LIN {X 0,Y 314.91,Z 685.03,A -85,B 0,C 180,E1 14211.742,E2 14211.742} C_VEL
LIN {X 0,Y 315.552,Z 685.03,A -85,B 0,C 180,E1 14220.006,E2 14220.006} C_VEL
LIN {X 0,Y 314.856,Z 685.03,A -85,B 0,C 180,E1 14228.272,E2 14228.272} C_VEL
LIN {X 0,Y 314.303,Z 685.03,A -85,B 0,C 180,E1 14236.747,E2 14236.747} C_VEL
LIN {X 0,Y 313.867,Z 685.03,A -85,B 0,C 180,E1 14244.013,E2 14244.013} C_VEL
LIN {X 0,Y 313.657,Z 685.474,A -85,B 0,C 180,E1 14251.561,E2 14251.561} C_VEL
LIN {X 0,Y 320.452,Z 702.79,A -85,B 0,C 180,E1 14254.351,E2 14254.351} C_VEL
LIN {X 0,Y 344.549,Z 753.186,A -85,B 0,C 180,E1 14259.732,E2 14259.732} C_VEL
LIN {X 0,Y 358.041,Z 788.652,A -85,B 0,C 180,E1 14263.338,E2 14263.338} C_VEL
LIN {X 0,Y 350.721,Z 828.357,A -85,B 0,C 180,E1 14265.87,E2 14265.87} C_VEL
LIN {X 0,Y 342.562,Z 865.255,A -85,B 0,C 180,E1 14269.272,E2 14269.272} C_VEL
LIN {X 0,Y 334.419,Z 899.619,A -85,B 0,C 180,E1 14273.687,E2 14273.687} C_VEL
LIN {X 0,Y 326.94,Z 930.331,A -85,B 0,C 180,E1 14279.119,E2 14279.119} C_VEL
LIN {X 0,Y 321.25,Z 955.655,A -85,B 0,C 180,E1 14285.339,E2 14285.339} C_VEL
LIN {X 0,Y 317.975,Z 973.935,A -85,B 0,C 180,E1 14291.651,E2 14291.651} C_VEL
LIN {X 0,Y 316.694,Z 986.498,A -85,B 0,C 180,E1 14298.102,E2 14298.102} C_VEL
LIN {X 0,Y 316.54,Z 993.494,A -85,B 0,C 180,E1 14304.533,E2 14304.533} C_VEL
LIN {X 0,Y 316.69,Z 995.183,A -85,B 0,C 180,E1 14310.004,E2 14310.004} C_VEL
LIN {X 0,Y 316.59,Z 992.89,A -85,B 0,C 180,E1 14315.475,E2 14315.475} C_VEL
LIN {X 0,Y 316.815,Z 985.329,A -85,B 0,C 180,E1 14321.838,E2 14321.838} C_VEL
LIN {X 0,Y 318.156,Z 971.681,A -85,B 0,C 180,E1 14328.447,E2 14328.447} C_VEL
LIN {X 0,Y 321.438,Z 951.786,A -85,B 0,C 180,E1 14334.999,E2 14334.999} C_VEL
LIN {X 0,Y 327.008,Z 926.051,A -85,B 0,C 180,E1 14341.158,E2 14341.158} C_VEL
LIN {X 0,Y 335.591,Z 892.049,A -85,B 0,C 180,E1 14347.18,E2 14347.18} C_VEL
LIN {X 0,Y 337.508,Z 885.124,A -85,B 0,C 180,E1 14348.196,E2 14348.196} C_VEL
LIN {X 0,Y 337.867,Z 872.8,A -85,B 0,C 180,E1 14350.32,E2 14350.32} C_VEL
LIN {X 0,Y 338.147,Z 861.845,A -85,B 0,C 180,E1 14352.148,E2 14352.148} C_VEL
LIN {X 0,Y 338.618,Z 860.138,A -85,B 0,C 180,E1 14352.366,E2 14352.366} C_VEL
LIN {X 0,Y 352.636,Z 816.47,A -85,B 0,C 180,E1 14356.882,E2 14356.882} C_VEL
LIN {X 0,Y 360.703,Z 791.738,A -85,B 0,C 180,E1 14358.863,E2 14358.863} C_VEL
LIN {X 0,Y 364.085,Z 771.223,A -85,B 0,C 180,E1 14361.96,E2 14361.96} C_VEL
LIN {X 0,Y 362.599,Z 769.841,A -85,B 0,C 180,E1 14364.361,E2 14364.361} C_VEL
LIN {X 0,Y 362.059,Z 771.868,A -85,B 0,C 180,E1 14366.312,E2 14366.312} C_VEL
LIN {X 0,Y 346.456,Z 811.757,A -85,B 0,C 180,E1 14369.757,E2 14369.757} C_VEL
LIN {X 0,Y 336.821,Z 840.977,A -85,B 0,C 180,E1 14373.38,E2 14373.38} C_VEL
LIN {X 0,Y 328.963,Z 862.947,A -85,B 0,C 180,E1 14377.403,E2 14377.403} C_VEL
LIN {X 0,Y 321.914,Z 880.59,A -85,B 0,C 180,E1 14382.256,E2 14382.256} C_VEL
LIN {X 0,Y 316.885,Z 891.625,A -85,B 0,C 180,E1 14387.145,E2 14387.145} C_VEL
LIN {X 0,Y 313.836,Z 897.239,A -85,B 0,C 180,E1 14391.701,E2 14391.701} C_VEL
LIN {X 0,Y 311.784,Z 898.859,A -85,B 0,C 180,E1 14397.22,E2 14397.22} C_VEL
LIN {X 0,Y 311.166,Z 894.893,A -85,B 0,C 180,E1 14402.773,E2 14402.773} C_VEL
LIN {X 0,Y 311.633,Z 885.117,A -85,B 0,C 180,E1 14408.346,E2 14408.346} C_VEL
LIN {X 0,Y 313.435,Z 869.481,A -85,B 0,C 180,E1 14413.567,E2 14413.567} C_VEL
LIN {X 0,Y 316.293,Z 848.979,A -85,B 0,C 180,E1 14418.112,E2 14418.112} C_VEL
LIN {X 0,Y 319.772,Z 823.229,A -85,B 0,C 180,E1 14421.989,E2 14421.989} C_VEL
LIN {X 0,Y 322.925,Z 794.302,A -85,B 0,C 180,E1 14424.861,E2 14424.861} C_VEL
LIN {X 0,Y 325.253,Z 762.343,A -85,B 0,C 180,E1 14426.77,E2 14426.77} C_VEL
LIN {X 0,Y 325.571,Z 741.227,A -85,B 0,C 180,E1 14427.634,E2 14427.634} C_VEL
LIN {X 0,Y 308.112,Z 692.452,A -85,B 0,C 180,E1 14431.358,E2 14431.358} C_VEL
LIN {X 0,Y 305.675,Z 685.03,A -85,B 0,C 180,E1 14432.04,E2 14432.04} C_VEL
LIN {X 0,Y 305.44,Z 685.03,A -85,B 0,C 180,E1 14439.948,E2 14439.948} C_VEL
LIN {X 0,Y 305.597,Z 685.776,A -85,B 0,C 180,E1 14445.292,E2 14445.292} C_VEL
LIN {X 0,Y 308.509,Z 691.107,A -85,B 0,C 180,E1 14446.016,E2 14446.016} C_VEL
LIN {X 0,Y 327.842,Z 726.86,A -85,B 0,C 180,E1 14450.419,E2 14450.419} C_VEL
LIN {X 0,Y 337.738,Z 754.456,A -85,B 0,C 180,E1 14453.52,E2 14453.52} C_VEL
LIN {X 0,Y 340.064,Z 767.182,A -85,B 0,C 180,E1 14454.899,E2 14454.899} C_VEL
LIN {X 0,Y 334.973,Z 797.319,A -85,B 0,C 180,E1 14457.653,E2 14457.653} C_VEL
LIN {X 0,Y 329.004,Z 824.07,A -85,B 0,C 180,E1 14461.239,E2 14461.239} C_VEL
LIN {X 0,Y 323.053,Z 846.325,A -85,B 0,C 180,E1 14465.482,E2 14465.482} C_VEL
LIN {X 0,Y 317.303,Z 865.927,A -85,B 0,C 180,E1 14470.911,E2 14470.911} C_VEL
LIN {X 0,Y 313.335,Z 879.686,A -85,B 0,C 180,E1 14476.771,E2 14476.771} C_VEL
LIN {X 0,Y 311.078,Z 888.192,A -85,B 0,C 180,E1 14483.03,E2 14483.03} C_VEL
LIN {X 0,Y 310.44,Z 891.269,A -85,B 0,C 180,E1 14489.996,E2 14489.996} C_VEL
LIN {X 0,Y 310.948,Z 888.611,A -85,B 0,C 180,E1 14496.334,E2 14496.334} C_VEL
LIN {X 0,Y 313.064,Z 880.748,A -85,B 0,C 180,E1 14502.524,E2 14502.524} C_VEL
LIN {X 0,Y 316.507,Z 868.508,A -85,B 0,C 180,E1 14508.075,E2 14508.075} C_VEL
LIN {X 0,Y 321.859,Z 850.589,A -85,B 0,C 180,E1 14513.391,E2 14513.391} C_VEL
LIN {X 0,Y 328.127,Z 827.373,A -85,B 0,C 180,E1 14518.114,E2 14518.114} C_VEL
LIN {X 0,Y 334.275,Z 800.831,A -85,B 0,C 180,E1 14521.841,E2 14521.841} C_VEL
LIN {X 0,Y 339.405,Z 771.117,A -85,B 0,C 180,E1 14524.694,E2 14524.694} C_VEL
LIN {X 0,Y 339.697,Z 763.15,A -85,B 0,C 180,E1 14525.388,E2 14525.388} C_VEL
LIN {X 0,Y 331.408,Z 735.367,A -85,B 0,C 180,E1 14528.517,E2 14528.517} C_VEL
LIN {X 0,Y 316.791,Z 705.665,A -85,B 0,C 180,E1 14531.941,E2 14531.941} C_VEL
LIN {X 0,Y 305.58,Z 685.941,A -85,B 0,C 180,E1 14534.578,E2 14534.578} C_VEL
LIN {X 0,Y 305.491,Z 685.03,A -85,B 0,C 180,E1 14534.816,E2 14534.816} C_VEL
LIN {X 0,Y 305.405,Z 685.03,A -85,B 0,C 180,E1 14542.234,E2 14542.234} C_VEL
LIN {X 0,Y 305.731,Z 685.03,A -85,B 0,C 180,E1 14550.434,E2 14550.434} C_VEL
LIN {X 0,Y 306.036,Z 685.03,A -85,B 0,C 180,E1 14556.776,E2 14556.776} C_VEL
LIN {X 0,Y 306.448,Z 685.03,A -85,B 0,C 180,E1 14562.824,E2 14562.824} C_VEL
LIN {X 0,Y 306.846,Z 685.03,A -85,B 0,C 180,E1 14569.588,E2 14569.588} C_VEL
LIN {X 0,Y 307.396,Z 685.03,A -85,B 0,C 180,E1 14577.193,E2 14577.193} C_VEL
LIN {X 0,Y 307.447,Z 685.03,A -85,B 0,C 180,E1 14582.819,E2 14582.819} C_VEL
LIN {X 0,Y 306.722,Z 685.03,A -85,B 0,C 180,E1 14591.355,E2 14591.355} C_VEL
LIN {X 0,Y 306.323,Z 685.03,A -85,B 0,C 180,E1 14597.197,E2 14597.197} C_VEL
LIN {X 0,Y 306.014,Z 685.03,A -85,B 0,C 180,E1 14603.239,E2 14603.239} C_VEL
LIN {X 0,Y 305.747,Z 685.427,A -85,B 0,C 180,E1 14610.369,E2 14610.369} C_VEL
LIN {X 0,Y 312.127,Z 701.796,A -85,B 0,C 180,E1 14613.058,E2 14613.058} C_VEL
LIN {X 0,Y 335.006,Z 749.372,A -85,B 0,C 180,E1 14618.375,E2 14618.375} C_VEL
LIN {X 0,Y 349.645,Z 785.813,A -85,B 0,C 180,E1 14622.259,E2 14622.259} C_VEL
LIN {X 0,Y 350.911,Z 791.551,A -85,B 0,C 180,E1 14622.803,E2 14622.803} C_VEL
LIN {X 0,Y 343.248,Z 831.026,A -85,B 0,C 180,E1 14625.448,E2 14625.448} C_VEL
LIN {X 0,Y 334.145,Z 870.49,A -85,B 0,C 180,E1 14629.31,E2 14629.31} C_VEL
LIN {X 0,Y 325.544,Z 905.238,A -85,B 0,C 180,E1 14634.136,E2 14634.136} C_VEL
LIN {X 0,Y 318.201,Z 934.458,A -85,B 0,C 180,E1 14639.747,E2 14639.747} C_VEL
LIN {X 0,Y 313.124,Z 956.64,A -85,B 0,C 180,E1 14645.558,E2 14645.558} C_VEL
LIN {X 0,Y 309.963,Z 974.481,A -85,B 0,C 180,E1 14652.092,E2 14652.092} C_VEL
LIN {X 0,Y 308.835,Z 986.462,A -85,B 0,C 180,E1 14658.733,E2 14658.733} C_VEL
LIN {X 0,Y 308.712,Z 992.233,A -85,B 0,C 180,E1 14664.394,E2 14664.394} C_VEL
LIN {X 0,Y 308.877,Z 993.977,A -85,B 0,C 180,E1 14670.004,E2 14670.004} C_VEL
LIN {X 0,Y 308.762,Z 991.696,A -85,B 0,C 180,E1 14675.614,E2 14675.614} C_VEL
LIN {X 0,Y 308.927,Z 985.403,A -85,B 0,C 180,E1 14681.272,E2 14681.272} C_VEL
LIN {X 0,Y 310.144,Z 972.746,A -85,B 0,C 180,E1 14687.957,E2 14687.957} C_VEL
LIN {X 0,Y 313.523,Z 952.562,A -85,B 0,C 180,E1 14695.05,E2 14695.05} C_VEL
LIN {X 0,Y 319.623,Z 926.044,A -85,B 0,C 180,E1 14701.694,E2 14701.694} C_VEL
LIN {X 0,Y 328.624,Z 892.919,A -85,B 0,C 180,E1 14707.805,E2 14707.805} C_VEL
LIN {X 0,Y 338.618,Z 860.138,A -85,B 0,C 180,E1 14712.366,E2 14712.366} C_VEL
LIN {X 0,Y 340.112,Z 847.359,A -85,B 0,C 180,E1 14714.385,E2 14714.385} C_VEL
LIN {X 0,Y 341.457,Z 836.061,A -85,B 0,C 180,E1 14716.115,E2 14716.115} C_VEL
LIN {X 0,Y 342.022,Z 834.288,A -85,B 0,C 180,E1 14716.308,E2 14716.308} C_VEL
LIN {X 0,Y 356.359,Z 794.468,A -85,B 0,C 180,E1 14719.879,E2 14719.879} C_VEL
LIN {X 0,Y 360.175,Z 777.996,A -85,B 0,C 180,E1 14722.415,E2 14722.415} C_VEL
LIN {X 0,Y 358.705,Z 777.781,A -85,B 0,C 180,E1 14725.392,E2 14725.392} C_VEL
LIN {X 0,Y 341.73,Z 816.303,A -85,B 0,C 180,E1 14728.926,E2 14728.926} C_VEL
LIN {X 0,Y 330.611,Z 845.629,A -85,B 0,C 180,E1 14732.839,E2 14732.839} C_VEL
LIN {X 0,Y 321.592,Z 868.061,A -85,B 0,C 180,E1 14737.32,E2 14737.32} C_VEL
LIN {X 0,Y 314.828,Z 883.244,A -85,B 0,C 180,E1 14741.842,E2 14741.842} C_VEL
LIN {X 0,Y 308.974,Z 894.716,A -85,B 0,C 180,E1 14747.442,E2 14747.442} C_VEL
LIN {X 0,Y 306.241,Z 899.036,A -85,B 0,C 180,E1 14751.493,E2 14751.493} C_VEL
LIN {X 0,Y 304.036,Z 900.353,A -85,B 0,C 180,E1 14757.149,E2 14757.149} C_VEL
LIN {X 0,Y 303.375,Z 896.076,A -85,B 0,C 180,E1 14762.844,E2 14762.844} C_VEL
LIN {X 0,Y 303.865,Z 885.986,A -85,B 0,C 180,E1 14768.561,E2 14768.561} C_VEL
LIN {X 0,Y 305.793,Z 870.096,A -85,B 0,C 180,E1 14773.912,E2 14773.912} C_VEL
LIN {X 0,Y 308.745,Z 849.486,A -85,B 0,C 180,E1 14778.515,E2 14778.515} C_VEL
LIN {X 0,Y 312.222,Z 824.404,A -85,B 0,C 180,E1 14782.363,E2 14782.363} C_VEL
LIN {X 0,Y 315.563,Z 795.059,A -85,B 0,C 180,E1 14785.351,E2 14785.351} C_VEL
LIN {X 0,Y 317.967,Z 763.242,A -85,B 0,C 180,E1 14787.294,E2 14787.294} C_VEL
LIN {X 0,Y 318.42,Z 743.378,A -85,B 0,C 180,E1 14788.13,E2 14788.13} C_VEL
LIN {X 0,Y 301.443,Z 695.733,A -85,B 0,C 180,E1 14791.889,E2 14791.889} C_VEL
LIN {X 0,Y 297.704,Z 685.03,A -85,B 0,C 180,E1 14792.842,E2 14792.842} C_VEL
LIN {X 0,Y 297.489,Z 685.03,A -85,B 0,C 180,E1 14801.243,E2 14801.243} C_VEL
LIN {X 0,Y 297.615,Z 685.594,A -85,B 0,C 180,E1 14803.689,E2 14803.689} C_VEL
LIN {X 0,Y 300.308,Z 690.958,A -85,B 0,C 180,E1 14804.426,E2 14804.426} C_VEL
LIN {X 0,Y 318.532,Z 722.999,A -85,B 0,C 180,E1 14808.791,E2 14808.791} C_VEL
LIN {X 0,Y 329.284,Z 749.961,A -85,B 0,C 180,E1 14811.961,E2 14811.961} C_VEL
LIN {X 0,Y 333.667,Z 768.812,A -85,B 0,C 180,E1 14814.162,E2 14814.162} C_VEL
LIN {X 0,Y 328.098,Z 800.011,A -85,B 0,C 180,E1 14817.086,E2 14817.086} C_VEL
LIN {X 0,Y 321.852,Z 826.592,A -85,B 0,C 180,E1 14820.786,E2 14820.786} C_VEL
LIN {X 0,Y 315.427,Z 849.445,A -85,B 0,C 180,E1 14825.336,E2 14825.336} C_VEL
LIN {X 0,Y 309.592,Z 868.194,A -85,B 0,C 180,E1 14830.786,E2 14830.786} C_VEL
LIN {X 0,Y 305.724,Z 880.935,A -85,B 0,C 180,E1 14836.436,E2 14836.436} C_VEL
LIN {X 0,Y 303.349,Z 889.437,A -85,B 0,C 180,E1 14842.851,E2 14842.851} C_VEL
LIN {X 0,Y 302.655,Z 892.514,A -85,B 0,C 180,E1 14849.996,E2 14849.996} C_VEL
LIN {X 0,Y 303.348,Z 889.351,A -85,B 0,C 180,E1 14857.14,E2 14857.14} C_VEL
LIN {X 0,Y 305.741,Z 880.768,A -85,B 0,C 180,E1 14863.555,E2 14863.555} C_VEL
LIN {X 0,Y 309.978,Z 866.893,A -85,B 0,C 180,E1 14869.55,E2 14869.55} C_VEL
LIN {X 0,Y 315.622,Z 848.688,A -85,B 0,C 180,E1 14874.741,E2 14874.741} C_VEL
LIN {X 0,Y 322.403,Z 824.257,A -85,B 0,C 180,E1 14879.497,E2 14879.497} C_VEL
LIN {X 0,Y 328.797,Z 796.311,A -85,B 0,C 180,E1 14883.218,E2 14883.218} C_VEL
LIN {X 0,Y 333.385,Z 766.458,A -85,B 0,C 180,E1 14885.976,E2 14885.976} C_VEL
LIN {X 0,Y 325.504,Z 738.984,A -85,B 0,C 180,E1 14889.205,E2 14889.205} C_VEL
LIN {X 0,Y 312.062,Z 710.888,A -85,B 0,C 180,E1 14892.592,E2 14892.592} C_VEL
LIN {X 0,Y 297.61,Z 685.828,A -85,B 0,C 180,E1 14896.172,E2 14896.172} C_VEL
LIN {X 0,Y 297.495,Z 685.03,A -85,B 0,C 180,E1 14904.247,E2 14904.247} C_VEL
LIN {X 0,Y 297.869,Z 685.03,A -85,B 0,C 180,E1 14912.884,E2 14912.884} C_VEL
LIN {X 0,Y 298.237,Z 685.03,A -85,B 0,C 180,E1 14919.265,E2 14919.265} C_VEL
LIN {X 0,Y 298.695,Z 685.03,A -85,B 0,C 180,E1 14925.377,E2 14925.377} C_VEL
LIN {X 0,Y 299.258,Z 685.03,A -85,B 0,C 180,E1 14934.219,E2 14934.219} C_VEL
LIN {X 0,Y 299.741,Z 685.03,A -85,B 0,C 180,E1 14940.006,E2 14940.006} C_VEL
LIN {X 0,Y 299.197,Z 685.03,A -85,B 0,C 180,E1 14945.795,E2 14945.795} C_VEL
LIN {X 0,Y 298.564,Z 685.03,A -85,B 0,C 180,E1 14954.643,E2 14954.643} C_VEL
LIN {X 0,Y 298.181,Z 685.03,A -85,B 0,C 180,E1 14960.752,E2 14960.752} C_VEL
LIN {X 0,Y 297.79,Z 685.414,A -85,B 0,C 180,E1 14969.13,E2 14969.13} C_VEL
LIN {X 0,Y 303.851,Z 700.84,A -85,B 0,C 180,E1 14971.748,E2 14971.748} C_VEL
LIN {X 0,Y 327.157,Z 749.096,A -85,B 0,C 180,E1 14977.364,E2 14977.364} C_VEL
LIN {X 0,Y 342.417,Z 787.359,A -85,B 0,C 180,E1 14981.593,E2 14981.593} C_VEL
LIN {X 0,Y 343.752,Z 794.393,A -85,B 0,C 180,E1 14982.257,E2 14982.257} C_VEL
LIN {X 0,Y 335.528,Z 834.821,A -85,B 0,C 180,E1 14985.131,E2 14985.131} C_VEL
LIN {X 0,Y 326.37,Z 872.454,A -85,B 0,C 180,E1 14989.009,E2 14989.009} C_VEL
LIN {X 0,Y 317.9,Z 905.743,A -85,B 0,C 180,E1 14993.803,E2 14993.803} C_VEL
LIN {X 0,Y 310.234,Z 935.287,A -85,B 0,C 180,E1 14999.695,E2 14999.695} C_VEL
LIN {X 0,Y 304.859,Z 958.008,A -85,B 0,C 180,E1 15005.973,E2 15005.973} C_VEL
LIN {X 0,Y 301.965,Z 974.875,A -85,B 0,C 180,E1 15012.556,E2 15012.556} C_VEL
LIN {X 0,Y 300.993,Z 985.055,A -85,B 0,C 180,E1 15018.436,E2 15018.436} C_VEL
LIN {X 0,Y 300.894,Z 990.951,A -85,B 0,C 180,E1 15024.248,E2 15024.248} C_VEL
LIN {X 0,Y 301.065,Z 992.763,A -85,B 0,C 180,E1 15030.004,E2 15030.004} C_VEL
LIN {X 0,Y 300.939,Z 990.492,A -85,B 0,C 180,E1 15035.76,E2 15035.76} C_VEL
LIN {X 0,Y 301.079,Z 984.177,A -85,B 0,C 180,E1 15041.57,E2 15041.57} C_VEL
LIN {X 0,Y 302.38,Z 971.295,A -85,B 0,C 180,E1 15048.521,E2 15048.521} C_VEL
LIN {X 0,Y 305.942,Z 951.774,A -85,B 0,C 180,E1 15055.574,E2 15055.574} C_VEL
LIN {X 0,Y 312.455,Z 925.457,A -85,B 0,C 180,E1 15062.401,E2 15062.401} C_VEL
LIN {X 0,Y 322.589,Z 891.375,A -85,B 0,C 180,E1 15068.88,E2 15068.88} C_VEL
LIN {X 0,Y 336.375,Z 850.113,A -85,B 0,C 180,E1 15074.583,E2 15074.583} C_VEL
LIN {X 0,Y 342.022,Z 834.288,A -85,B 0,C 180,E1 15076.308,E2 15076.308} C_VEL
LIN {X 0,Y 344.91,Z 821.142,A -85,B 0,C 180,E1 15078.186,E2 15078.186} C_VEL
LIN {X 0,Y 348.257,Z 807.865,A -85,B 0,C 180,E1 15079.98,E2 15079.98} C_VEL
LIN {X 0,Y 352.562,Z 796.568,A -85,B 0,C 180,E1 15081.045,E2 15081.045} C_VEL
LIN {X 0,Y 356.225,Z 784.754,A -85,B 0,C 180,E1 15082.866,E2 15082.866} C_VEL
LIN {X 0,Y 355.329,Z 784.395,A -85,B 0,C 180,E1 15084.529,E2 15084.529} C_VEL
LIN {X 0,Y 337.166,Z 821.047,A -85,B 0,C 180,E1 15088.08,E2 15088.08} C_VEL
LIN {X 0,Y 325.143,Z 848.745,A -85,B 0,C 180,E1 15092.005,E2 15092.005} C_VEL
LIN {X 0,Y 315.667,Z 869.856,A -85,B 0,C 180,E1 15096.395,E2 15096.395} C_VEL
LIN {X 0,Y 307.77,Z 885.885,A -85,B 0,C 180,E1 15101.411,E2 15101.411} C_VEL
LIN {X 0,Y 301.692,Z 896.612,A -85,B 0,C 180,E1 15106.987,E2 15106.987} C_VEL
LIN {X 0,Y 298.639,Z 900.848,A -85,B 0,C 180,E1 15111.275,E2 15111.275} C_VEL
LIN {X 0,Y 296.282,Z 901.811,A -85,B 0,C 180,E1 15117.074,E2 15117.074} C_VEL
LIN {X 0,Y 295.585,Z 897.235,A -85,B 0,C 180,E1 15122.92,E2 15122.92} C_VEL
LIN {X 0,Y 295.948,Z 888.486,A -85,B 0,C 180,E1 15128.053,E2 15128.053} C_VEL
LIN {X 0,Y 297.771,Z 873.182,A -85,B 0,C 180,E1 15133.547,E2 15133.547} C_VEL
LIN {X 0,Y 300.658,Z 853.477,A -85,B 0,C 180,E1 15138.273,E2 15138.273} C_VEL
LIN {X 0,Y 304.329,Z 828.2,A -85,B 0,C 180,E1 15142.398,E2 15142.398} C_VEL
LIN {X 0,Y 307.827,Z 799.113,A -85,B 0,C 180,E1 15145.569,E2 15145.569} C_VEL
LIN {X 0,Y 310.479,Z 767.633,A -85,B 0,C 180,E1 15147.675,E2 15147.675} C_VEL
LIN {X 0,Y 311.047,Z 744.671,A -85,B 0,C 180,E1 15148.7,E2 15148.7} C_VEL
LIN {X 0,Y 293.605,Z 695.813,A -85,B 0,C 180,E1 15152.732,E2 15152.732} C_VEL
LIN {X 0,Y 289.657,Z 685.03,A -85,B 0,C 180,E1 15153.855,E2 15153.855} C_VEL
LIN {X 0,Y 289.583,Z 685.411,A -85,B 0,C 180,E1 15161.931,E2 15161.931} C_VEL
LIN {X 0,Y 292.1,Z 690.804,A -85,B 0,C 180,E1 15162.693,E2 15162.693} C_VEL
LIN {X 0,Y 308.6,Z 718.15,A -85,B 0,C 180,E1 15166.899,E2 15166.899} C_VEL
LIN {X 0,Y 320.84,Z 745.773,A -85,B 0,C 180,E1 15170.353,E2 15170.353} C_VEL
LIN {X 0,Y 327.286,Z 770.35,A -85,B 0,C 180,E1 15173.383,E2 15173.383} C_VEL
LIN {X 0,Y 321.591,Z 801.234,A -85,B 0,C 180,E1 15176.332,E2 15176.332} C_VEL
LIN {X 0,Y 315.11,Z 827.625,A -85,B 0,C 180,E1 15180.058,E2 15180.058} C_VEL
LIN {X 0,Y 308.351,Z 850.686,A -85,B 0,C 180,E1 15184.731,E2 15184.731} C_VEL
LIN {X 0,Y 302.218,Z 869.44,A -85,B 0,C 180,E1 15190.298,E2 15190.298} C_VEL
LIN {X 0,Y 297.784,Z 883.416,A -85,B 0,C 180,E1 15196.813,E2 15196.813} C_VEL
LIN {X 0,Y 295.601,Z 890.685,A -85,B 0,C 180,E1 15202.663,E2 15202.663} C_VEL
LIN {X 0,Y 294.864,Z 893.76,A -85,B 0,C 180,E1 15209.996,E2 15209.996} C_VEL
LIN {X 0,Y 295.601,Z 890.6,A -85,B 0,C 180,E1 15217.328,E2 15217.328} C_VEL
LIN {X 0,Y 298.144,Z 882.019,A -85,B 0,C 180,E1 15223.907,E2 15223.907} C_VEL
LIN {X 0,Y 302.632,Z 868.14,A -85,B 0,C 180,E1 15230.044,E2 15230.044} C_VEL
LIN {X 0,Y 308.551,Z 849.934,A -85,B 0,C 180,E1 15235.347,E2 15235.347} C_VEL
LIN {X 0,Y 315.542,Z 825.812,A -85,B 0,C 180,E1 15240.143,E2 15240.143} C_VEL
LIN {X 0,Y 322.323,Z 797.543,A -85,B 0,C 180,E1 15243.975,E2 15243.975} C_VEL
LIN {X 0,Y 326.938,Z 768.812,A -85,B 0,C 180,E1 15246.7,E2 15246.7} C_VEL
LIN {X 0,Y 319.406,Z 741.93,A -85,B 0,C 180,E1 15249.998,E2 15249.998} C_VEL
LIN {X 0,Y 306.159,Z 713.961,A -85,B 0,C 180,E1 15253.554,E2 15253.554} C_VEL
LIN {X 0,Y 291.571,Z 690.291,A -85,B 0,C 180,E1 15257.307,E2 15257.307} C_VEL
LIN {X 0,Y 289.534,Z 685.03,A -85,B 0,C 180,E1 15258.057,E2 15258.057} C_VEL
LIN {X 0,Y 289.659,Z 685.03,A -85,B 0,C 180,E1 15266.46,E2 15266.46} C_VEL
LIN {X 0,Y 289.863,Z 685.03,A -85,B 0,C 180,E1 15272.248,E2 15272.248} C_VEL
LIN {X 0,Y 290.34,Z 685.03,A -85,B 0,C 180,E1 15279.308,E2 15279.308} C_VEL
LIN {X 0,Y 290.918,Z 685.03,A -85,B 0,C 180,E1 15288.033,E2 15288.033} C_VEL
LIN {X 0,Y 291.57,Z 685.03,A -85,B 0,C 180,E1 15297.04,E2 15297.04} C_VEL
LIN {X 0,Y 291.623,Z 685.03,A -85,B 0,C 180,E1 15302.972,E2 15302.972} C_VEL
LIN {X 0,Y 290.813,Z 685.03,A -85,B 0,C 180,E1 15311.985,E2 15311.985} C_VEL
LIN {X 0,Y 290.286,Z 685.03,A -85,B 0,C 180,E1 15320.664,E2 15320.664} C_VEL
LIN {X 0,Y 289.886,Z 685.383,A -85,B 0,C 180,E1 15327.858,E2 15327.858} C_VEL
LIN {X 0,Y 295.63,Z 699.896,A -85,B 0,C 180,E1 15330.378,E2 15330.378} C_VEL
LIN {X 0,Y 319.22,Z 748.898,A -85,B 0,C 180,E1 15336.314,E2 15336.314} C_VEL
LIN {X 0,Y 334.247,Z 786.346,A -85,B 0,C 180,E1 15340.62,E2 15340.62} C_VEL
LIN {X 0,Y 336.831,Z 795.847,A -85,B 0,C 180,E1 15341.63,E2 15341.63} C_VEL
LIN {X 0,Y 328.33,Z 835.744,A -85,B 0,C 180,E1 15344.574,E2 15344.574} C_VEL
LIN {X 0,Y 318.983,Z 872.969,A -85,B 0,C 180,E1 15348.528,E2 15348.528} C_VEL
LIN {X 0,Y 310.308,Z 905.886,A -85,B 0,C 180,E1 15353.412,E2 15353.412} C_VEL
LIN {X 0,Y 302.588,Z 934.769,A -85,B 0,C 180,E1 15359.331,E2 15359.331} C_VEL
LIN {X 0,Y 296.902,Z 958.133,A -85,B 0,C 180,E1 15366.012,E2 15366.012} C_VEL
LIN {X 0,Y 294.026,Z 974.803,A -85,B 0,C 180,E1 15372.84,E2 15372.84} C_VEL
LIN {X 0,Y 293.098,Z 985.518,A -85,B 0,C 180,E1 15379.623,E2 15379.623} C_VEL
LIN {X 0,Y 293.067,Z 989.642,A -85,B 0,C 180,E1 15384.093,E2 15384.093} C_VEL
LIN {X 0,Y 293.277,Z 991.533,A -85,B 0,C 180,E1 15390.004,E2 15390.004} C_VEL
LIN {X 0,Y 293.107,Z 989.281,A -85,B 0,C 180,E1 15395.915,E2 15395.915} C_VEL
LIN {X 0,Y 293.243,Z 982.642,A -85,B 0,C 180,E1 15402.109,E2 15402.109} C_VEL
LIN {X 0,Y 294.6,Z 970.061,A -85,B 0,C 180,E1 15409.029,E2 15409.029} C_VEL
LIN {X 0,Y 298.476,Z 950.64,A -85,B 0,C 180,E1 15416.262,E2 15416.262} C_VEL
LIN {X 0,Y 305.6,Z 924.187,A -85,B 0,C 180,E1 15423.328,E2 15423.328} C_VEL
LIN {X 0,Y 317.038,Z 889.177,A -85,B 0,C 180,E1 15430.152,E2 15430.152} C_VEL
LIN {X 0,Y 332.242,Z 848.034,A -85,B 0,C 180,E1 15435.934,E2 15435.934} C_VEL
LIN {X 0,Y 348.257,Z 807.865,A -85,B 0,C 180,E1 15439.98,E2 15439.98} C_VEL
LIN {X 0,Y 349.723,Z 801.928,A -85,B 0,C 180,E1 15440.992,E2 15440.992} C_VEL
LIN {X 0,Y 351.205,Z 793.819,A -85,B 0,C 180,E1 15443.07,E2 15443.07} C_VEL
LIN {X 0,Y 352.109,Z 791.279,A -85,B 0,C 180,E1 15443.661,E2 15443.661} C_VEL
LIN {X 0,Y 333.305,Z 824.909,A -85,B 0,C 180,E1 15447.089,E2 15447.089} C_VEL
LIN {X 0,Y 319.803,Z 852.079,A -85,B 0,C 180,E1 15451.148,E2 15451.148} C_VEL
LIN {X 0,Y 309.08,Z 873.383,A -85,B 0,C 180,E1 15455.86,E2 15455.86} C_VEL
LIN {X 0,Y 300.743,Z 888.568,A -85,B 0,C 180,E1 15460.96,E2 15460.96} C_VEL
LIN {X 0,Y 294.296,Z 898.743,A -85,B 0,C 180,E1 15466.655,E2 15466.655} C_VEL
LIN {X 0,Y 291.054,Z 902.684,A -85,B 0,C 180,E1 15471.046,E2 15471.046} C_VEL
LIN {X 0,Y 288.535,Z 903.253,A -85,B 0,C 180,E1 15476.996,E2 15476.996} C_VEL
LIN {X 0,Y 287.794,Z 898.384,A -85,B 0,C 180,E1 15482.999,E2 15482.999} C_VEL
LIN {X 0,Y 288.333,Z 887.636,A -85,B 0,C 180,E1 15489.026,E2 15489.026} C_VEL
LIN {X 0,Y 290.286,Z 872.444,A -85,B 0,C 180,E1 15494.287,E2 15494.287} C_VEL
LIN {X 0,Y 293.428,Z 851.706,A -85,B 0,C 180,E1 15499.129,E2 15499.129} C_VEL
LIN {X 0,Y 297.186,Z 826.62,A -85,B 0,C 180,E1 15503.164,E2 15503.164} C_VEL
LIN {X 0,Y 300.739,Z 797.348,A -85,B 0,C 180,E1 15506.3,E2 15506.3} C_VEL
LIN {X 0,Y 303.382,Z 765.088,A -85,B 0,C 180,E1 15508.388,E2 15508.388} C_VEL
LIN {X 0,Y 303.815,Z 746.49,A -85,B 0,C 180,E1 15509.245,E2 15509.245} C_VEL
LIN {X 0,Y 286.357,Z 697.38,A -85,B 0,C 180,E1 15513.469,E2 15513.469} C_VEL
LIN {X 0,Y 281.715,Z 685.03,A -85,B 0,C 180,E1 15514.801,E2 15514.801} C_VEL
LIN {X 0,Y 281.711,Z 685.822,A -85,B 0,C 180,E1 15520.067,E2 15520.067} C_VEL
LIN {X 0,Y 284.697,Z 691.263,A -85,B 0,C 180,E1 15521.01,E2 15521.01} C_VEL
LIN {X 0,Y 302.327,Z 720.548,A -85,B 0,C 180,E1 15525.817,E2 15525.817} C_VEL
LIN {X 0,Y 314.306,Z 747.295,A -85,B 0,C 180,E1 15529.376,E2 15529.376} C_VEL
LIN {X 0,Y 320.914,Z 772.646,A -85,B 0,C 180,E1 15532.647,E2 15532.647} C_VEL
LIN {X 0,Y 315.136,Z 802.459,A -85,B 0,C 180,E1 15535.547,E2 15535.547} C_VEL
LIN {X 0,Y 308.032,Z 830.111,A -85,B 0,C 180,E1 15539.553,E2 15539.553} C_VEL
LIN {X 0,Y 300.702,Z 853.744,A -85,B 0,C 180,E1 15544.568,E2 15544.568} C_VEL
LIN {X 0,Y 294.883,Z 870.683,A -85,B 0,C 180,E1 15549.787,E2 15549.787} C_VEL
LIN {X 0,Y 290.549,Z 883.43,A -85,B 0,C 180,E1 15555.712,E2 15555.712} C_VEL
LIN {X 0,Y 287.878,Z 891.93,A -85,B 0,C 180,E1 15562.465,E2 15562.465} C_VEL
LIN {X 0,Y 287.149,Z 894.491,A -85,B 0,C 180,E1 15566.983,E2 15566.983} C_VEL
LIN {X 0,Y 287.172,Z 894.326,A -85,B 0,C 180,E1 15573.449,E2 15573.449} C_VEL
LIN {X 0,Y 288.835,Z 888.712,A -85,B 0,C 180,E1 15580.532,E2 15580.532} C_VEL
LIN {X 0,Y 292.627,Z 877.21,A -85,B 0,C 180,E1 15587.386,E2 15587.386} C_VEL
LIN {X 0,Y 298.418,Z 860.49,A -85,B 0,C 180,E1 15593.463,E2 15593.463} C_VEL
LIN {X 0,Y 305.508,Z 838.482,A -85,B 0,C 180,E1 15598.786,E2 15598.786} C_VEL
LIN {X 0,Y 312.752,Z 812.39,A -85,B 0,C 180,E1 15603.077,E2 15603.077} C_VEL
LIN {X 0,Y 319.082,Z 782.905,A -85,B 0,C 180,E1 15606.374,E2 15606.374} C_VEL
LIN {X 0,Y 320.633,Z 771.591,A -85,B 0,C 180,E1 15607.392,E2 15607.392} C_VEL
LIN {X 0,Y 313.14,Z 744.192,A -85,B 0,C 180,E1 15610.905,E2 15610.905} C_VEL
LIN {X 0,Y 300.403,Z 717.207,A -85,B 0,C 180,E1 15614.538,E2 15614.538} C_VEL
LIN {X 0,Y 284.194,Z 690.862,A -85,B 0,C 180,E1 15618.985,E2 15618.985} C_VEL
LIN {X 0,Y 281.738,Z 685.987,A -85,B 0,C 180,E1 15619.777,E2 15619.777} C_VEL
LIN {X 0,Y 281.639,Z 685.03,A -85,B 0,C 180,E1 15620.001,E2 15620.001} C_VEL
LIN {X 0,Y 281.762,Z 685.03,A -85,B 0,C 180,E1 15628.965,E2 15628.965} C_VEL
LIN {X 0,Y 282.213,Z 685.03,A -85,B 0,C 180,E1 15638.029,E2 15638.029} C_VEL
LIN {X 0,Y 282.739,Z 685.03,A -85,B 0,C 180,E1 15644.531,E2 15644.531} C_VEL
LIN {X 0,Y 283.227,Z 685.03,A -85,B 0,C 180,E1 15652.921,E2 15652.921} C_VEL
LIN {X 0,Y 283.929,Z 685.03,A -85,B 0,C 180,E1 15660.007,E2 15660.007} C_VEL
LIN {X 0,Y 283.33,Z 685.03,A -85,B 0,C 180,E1 15666.121,E2 15666.121} C_VEL
LIN {X 0,Y 282.845,Z 685.03,A -85,B 0,C 180,E1 15672.328,E2 15672.328} C_VEL
LIN {X 0,Y 282.408,Z 685.03,A -85,B 0,C 180,E1 15678.705,E2 15678.705} C_VEL
LIN {X 0,Y 281.951,Z 685.284,A -85,B 0,C 180,E1 15686.52,E2 15686.52} C_VEL
LIN {X 0,Y 287.386,Z 698.972,A -85,B 0,C 180,E1 15688.956,E2 15688.956} C_VEL
LIN {X 0,Y 311.231,Z 748.305,A -85,B 0,C 180,E1 15695.204,E2 15695.204} C_VEL
LIN {X 0,Y 326.789,Z 787.205,A -85,B 0,C 180,E1 15699.848,E2 15699.848} C_VEL
LIN {X 0,Y 329.716,Z 798.014,A -85,B 0,C 180,E1 15701.046,E2 15701.046} C_VEL
LIN {X 0,Y 321.174,Z 836.533,A -85,B 0,C 180,E1 15703.994,E2 15703.994} C_VEL
LIN {X 0,Y 311.719,Z 872.923,A -85,B 0,C 180,E1 15707.97,E2 15707.97} C_VEL
LIN {X 0,Y 302.766,Z 905.862,A -85,B 0,C 180,E1 15712.987,E2 15712.987} C_VEL
LIN {X 0,Y 295.03,Z 933.832,A -85,B 0,C 180,E1 15718.87,E2 15718.87} C_VEL
LIN {X 0,Y 289.13,Z 957.328,A -85,B 0,C 180,E1 15725.757,E2 15725.757} C_VEL
LIN {X 0,Y 286.271,Z 973.122,A -85,B 0,C 180,E1 15732.36,E2 15732.36} C_VEL
LIN {X 0,Y 285.282,Z 984.161,A -85,B 0,C 180,E1 15739.409,E2 15739.409} C_VEL
LIN {X 0,Y 285.274,Z 988.308,A -85,B 0,C 180,E1 15743.931,E2 15743.931} C_VEL
LIN {X 0,Y 285.475,Z 990.285,A -85,B 0,C 180,E1 15750.005,E2 15750.005} C_VEL
LIN {X 0,Y 285.268,Z 988.075,A -85,B 0,C 180,E1 15756.078,E2 15756.078} C_VEL
LIN {X 0,Y 285.442,Z 980.664,A -85,B 0,C 180,E1 15762.989,E2 15762.989} C_VEL
LIN {X 0,Y 286.967,Z 968.298,A -85,B 0,C 180,E1 15769.832,E2 15769.832} C_VEL
LIN {X 0,Y 291.048,Z 949.579,A -85,B 0,C 180,E1 15776.985,E2 15776.985} C_VEL
LIN {X 0,Y 298.715,Z 923.504,A -85,B 0,C 180,E1 15784.201,E2 15784.201} C_VEL
LIN {X 0,Y 311.295,Z 888.365,A -85,B 0,C 180,E1 15791.285,E2 15791.285} C_VEL
LIN {X 0,Y 328.461,Z 846.504,A -85,B 0,C 180,E1 15797.322,E2 15797.322} C_VEL
LIN {X 0,Y 347.557,Z 803.523,A -85,B 0,C 180,E1 15801.614,E2 15801.614} C_VEL
LIN {X 0,Y 351.205,Z 793.819,A -85,B 0,C 180,E1 15803.07,E2 15803.07} C_VEL
LIN {X 0,Y 349.901,Z 795.468,A -85,B 0,C 180,E1 15803.567,E2 15803.567} C_VEL
LIN {X 0,Y 339.331,Z 813.098,A -85,B 0,C 180,E1 15804.231,E2 15804.231} C_VEL
LIN {X 0,Y 321.505,Z 843.33,A -85,B 0,C 180,E1 15808.124,E2 15808.124} C_VEL
LIN {X 0,Y 307.469,Z 868.341,A -85,B 0,C 180,E1 15812.997,E2 15812.997} C_VEL
LIN {X 0,Y 296.971,Z 886.25,A -85,B 0,C 180,E1 15818.378,E2 15818.378} C_VEL
LIN {X 0,Y 289.11,Z 897.998,A -85,B 0,C 180,E1 15824.091,E2 15824.091} C_VEL
LIN {X 0,Y 284.333,Z 903.818,A -85,B 0,C 180,E1 15829.556,E2 15829.556} C_VEL
LIN {X 0,Y 281.97,Z 905.242,A -85,B 0,C 180,E1 15833.849,E2 15833.849} C_VEL
LIN {X 0,Y 280.373,Z 902.753,A -85,B 0,C 180,E1 15839.993,E2 15839.993} C_VEL
LIN {X 0,Y 280.073,Z 894.75,A -85,B 0,C 180,E1 15846.179,E2 15846.179} C_VEL
LIN {X 0,Y 281.423,Z 881.426,A -85,B 0,C 180,E1 15851.984,E2 15851.984} C_VEL
LIN {X 0,Y 284.32,Z 861.887,A -85,B 0,C 180,E1 15857.51,E2 15857.51} C_VEL
LIN {X 0,Y 288.107,Z 837.78,A -85,B 0,C 180,E1 15862.105,E2 15862.105} C_VEL
LIN {X 0,Y 291.852,Z 810.872,A -85,B 0,C 180,E1 15865.605,E2 15865.605} C_VEL
LIN {X 0,Y 295.133,Z 779.965,A -85,B 0,C 180,E1 15868.192,E2 15868.192} C_VEL
LIN {X 0,Y 296.69,Z 748.766,A -85,B 0,C 180,E1 15869.78,E2 15869.78} C_VEL
LIN {X 0,Y 279.981,Z 701.251,A -85,B 0,C 180,E1 15874.001,E2 15874.001} C_VEL
LIN {X 0,Y 273.682,Z 685.03,A -85,B 0,C 180,E1 15875.872,E2 15875.872} C_VEL
LIN {X 0,Y 273.567,Z 685.03,A -85,B 0,C 180,E1 15877.872,E2 15877.872} C_VEL
LIN {X 0,Y 275.838,Z 690.531,A -85,B 0,C 180,E1 15878.737,E2 15878.737} C_VEL
LIN {X 0,Y 282.135,Z 699.697,A -85,B 0,C 180,E1 15880.718,E2 15880.718} C_VEL
LIN {X 0,Y 298.098,Z 726.566,A -85,B 0,C 180,E1 15885.235,E2 15885.235} C_VEL
LIN {X 0,Y 308.936,Z 752.364,A -85,B 0,C 180,E1 15888.821,E2 15888.821} C_VEL
LIN {X 0,Y 314.426,Z 776.099,A -85,B 0,C 180,E1 15891.981,E2 15891.981} C_VEL
LIN {X 0,Y 308.113,Z 806.451,A -85,B 0,C 180,E1 15895.075,E2 15895.075} C_VEL
LIN {X 0,Y 300.566,Z 833.959,A -85,B 0,C 180,E1 15899.265,E2 15899.265} C_VEL
LIN {X 0,Y 293.058,Z 856.76,A -85,B 0,C 180,E1 15904.384,E2 15904.384} C_VEL
LIN {X 0,Y 286.877,Z 873.809,A -85,B 0,C 180,E1 15910.001,E2 15910.001} C_VEL
LIN {X 0,Y 282.562,Z 885.916,A -85,B 0,C 180,E1 15916.089,E2 15916.089} C_VEL
LIN {X 0,Y 280.151,Z 893.175,A -85,B 0,C 180,E1 15922.256,E2 15922.256} C_VEL
LIN {X 0,Y 279.285,Z 896.252,A -85,B 0,C 180,E1 15929.995,E2 15929.995} C_VEL
LIN {X 0,Y 280.154,Z 893.093,A -85,B 0,C 180,E1 15937.735,E2 15937.735} C_VEL
LIN {X 0,Y 283.008,Z 884.517,A -85,B 0,C 180,E1 15944.667,E2 15944.667} C_VEL
LIN {X 0,Y 288.004,Z 870.638,A -85,B 0,C 180,E1 15951.11,E2 15951.11} C_VEL
LIN {X 0,Y 294.672,Z 851.943,A -85,B 0,C 180,E1 15956.766,E2 15956.766} C_VEL
LIN {X 0,Y 302.468,Z 827.292,A -85,B 0,C 180,E1 15961.802,E2 15961.802} C_VEL
LIN {X 0,Y 309.527,Z 800.012,A -85,B 0,C 180,E1 15965.587,E2 15965.587} C_VEL
LIN {X 0,Y 314.356,Z 774.663,A -85,B 0,C 180,E1 15968.069,E2 15968.069} C_VEL
LIN {X 0,Y 307.217,Z 747.369,A -85,B 0,C 180,E1 15971.742,E2 15971.742} C_VEL
LIN {X 0,Y 294.594,Z 720.159,A -85,B 0,C 180,E1 15975.6,E2 15975.6} C_VEL
LIN {X 0,Y 279.366,Z 695.708,A -85,B 0,C 180,E1 15979.986,E2 15979.986} C_VEL
LIN {X 0,Y 275.787,Z 690.47,A -85,B 0,C 180,E1 15981.131,E2 15981.131} C_VEL
LIN {X 0,Y 273.55,Z 685.03,A -85,B 0,C 180,E1 15982.112,E2 15982.112} C_VEL
LIN {X 0,Y 273.866,Z 685.03,A -85,B 0,C 180,E1 15990.282,E2 15990.282} C_VEL
LIN {X 0,Y 274.308,Z 685.03,A -85,B 0,C 180,E1 15999.253,E2 15999.253} C_VEL
LIN {X 0,Y 275.012,Z 685.03,A -85,B 0,C 180,E1 16007.33,E2 16007.33} C_VEL
LIN {X 0,Y 275.448,Z 685.03,A -85,B 0,C 180,E1 16013.717,E2 16013.717} C_VEL
LIN {X 0,Y 276.022,Z 685.03,A -85,B 0,C 180,E1 16020.007,E2 16020.007} C_VEL
LIN {X 0,Y 275.39,Z 685.03,A -85,B 0,C 180,E1 16026.298,E2 16026.298} C_VEL
LIN {X 0,Y 274.89,Z 685.03,A -85,B 0,C 180,E1 16032.69,E2 16032.69} C_VEL
LIN {X 0,Y 274.279,Z 685.03,A -85,B 0,C 180,E1 16040.731,E2 16040.731} C_VEL
LIN {X 0,Y 274.134,Z 685.529,A -85,B 0,C 180,E1 16045.2,E2 16045.2} C_VEL
LIN {X 0,Y 279.107,Z 698.033,A -85,B 0,C 180,E1 16047.473,E2 16047.473} C_VEL
LIN {X 0,Y 302.675,Z 746.502,A -85,B 0,C 180,E1 16053.905,E2 16053.905} C_VEL
LIN {X 0,Y 318.662,Z 786.235,A -85,B 0,C 180,E1 16058.829,E2 16058.829} C_VEL
LIN {X 0,Y 322.778,Z 798.298,A -85,B 0,C 180,E1 16060.312,E2 16060.312} C_VEL
LIN {X 0,Y 313.954,Z 837.522,A -85,B 0,C 180,E1 16063.429,E2 16063.429} C_VEL
LIN {X 0,Y 303.976,Z 874.709,A -85,B 0,C 180,E1 16067.642,E2 16067.642} C_VEL
LIN {X 0,Y 294.543,Z 908.168,A -85,B 0,C 180,E1 16072.992,E2 16072.992} C_VEL
LIN {X 0,Y 286.401,Z 936.747,A -85,B 0,C 180,E1 16079.405,E2 16079.405} C_VEL
LIN {X 0,Y 280.904,Z 958.767,A -85,B 0,C 180,E1 16086.347,E2 16086.347} C_VEL
LIN {X 0,Y 278.185,Z 974.421,A -85,B 0,C 180,E1 16093.479,E2 16093.479} C_VEL
LIN {X 0,Y 277.411,Z 984.311,A -85,B 0,C 180,E1 16100.612,E2 16100.612} C_VEL
LIN {X 0,Y 277.501,Z 988.502,A -85,B 0,C 180,E1 16106.887,E2 16106.887} C_VEL
LIN {X 0,Y 277.687,Z 989.03,A -85,B 0,C 180,E1 16110.005,E2 16110.005} C_VEL
LIN {X 0,Y 277.436,Z 986.858,A -85,B 0,C 180,E1 16116.25,E2 16116.25} C_VEL
LIN {X 0,Y 277.597,Z 979.474,A -85,B 0,C 180,E1 16123.363,E2 16123.363} C_VEL
LIN {X 0,Y 279.377,Z 966.832,A -85,B 0,C 180,E1 16130.56,E2 16130.56} C_VEL
LIN {X 0,Y 284.371,Z 946.229,A -85,B 0,C 180,E1 16138.534,E2 16138.534} C_VEL
LIN {X 0,Y 293.69,Z 918.317,A -85,B 0,C 180,E1 16146.227,E2 16146.227} C_VEL
LIN {X 0,Y 307.973,Z 882.851,A -85,B 0,C 180,E1 16153.321,E2 16153.321} C_VEL
LIN {X 0,Y 326.736,Z 842.093,A -85,B 0,C 180,E1 16159.146,E2 16159.146} C_VEL
LIN {X 0,Y 345.376,Z 804.222,A -85,B 0,C 180,E1 16162.993,E2 16162.993} C_VEL
LIN {X 0,Y 345.969,Z 802.844,A -85,B 0,C 180,E1 16163.235,E2 16163.235} C_VEL
LIN {X 0,Y 339.331,Z 813.098,A -85,B 0,C 180,E1 16164.231,E2 16164.231} C_VEL
LIN {X 0,Y 336.407,Z 818.105,A -85,B 0,C 180,E1 16164.084,E2 16164.084} C_VEL
LIN {X 0,Y 330.276,Z 830.129,A -85,B 0,C 180,E1 16161.874,E2 16161.874} C_VEL
LIN {X 0,Y 309.198,Z 869.912,A -85,B 0,C 180,E1 16156.689,E2 16156.689} C_VEL
LIN {X 0,Y 291.777,Z 906.903,A -85,B 0,C 180,E1 16149.801,E2 16149.801} C_VEL
LIN {X 0,Y 280.098,Z 936.807,A -85,B 0,C 180,E1 16142.103,E2 16142.103} C_VEL
LIN {X 0,Y 273.094,Z 959.905,A -85,B 0,C 180,E1 16133.842,E2 16133.842} C_VEL
LIN {X 0,Y 270.155,Z 974.687,A -85,B 0,C 180,E1 16126.223,E2 16126.223} C_VEL
LIN {X 0,Y 269.582,Z 983.002,A -85,B 0,C 180,E1 16119.673,E2 16119.673} C_VEL
LIN {X 0,Y 269.658,Z 987.182,A -85,B 0,C 180,E1 16113.213,E2 16113.213} C_VEL
LIN {X 0,Y 269.911,Z 987.746,A -85,B 0,C 180,E1 16110.005,E2 16110.005} C_VEL
LIN {X 0,Y 269.666,Z 985.554,A -85,B 0,C 180,E1 16103.579,E2 16103.579} C_VEL
LIN {X 0,Y 269.848,Z 977.876,A -85,B 0,C 180,E1 16096.256,E2 16096.256} C_VEL
LIN {X 0,Y 271.781,Z 964.439,A -85,B 0,C 180,E1 16088.849,E2 16088.849} C_VEL
LIN {X 0,Y 276.439,Z 944.479,A -85,B 0,C 180,E1 16081.473,E2 16081.473} C_VEL
LIN {X 0,Y 283.889,Z 918.129,A -85,B 0,C 180,E1 16074.638,E2 16074.638} C_VEL
LIN {X 0,Y 293.337,Z 886.308,A -85,B 0,C 180,E1 16068.771,E2 16068.771} C_VEL
LIN {X 0,Y 303.492,Z 850.476,A -85,B 0,C 180,E1 16064.085,E2 16064.085} C_VEL
LIN {X 0,Y 313.182,Z 811.673,A -85,B 0,C 180,E1 16060.517,E2 16060.517} C_VEL
LIN {X 0,Y 315.243,Z 799.118,A -85,B 0,C 180,E1 16059.543,E2 16059.543} C_VEL
LIN {X 0,Y 301.273,Z 761.794,A -85,B 0,C 180,E1 16054.737,E2 16054.737} C_VEL
LIN {X 0,Y 282.702,Z 720.798,A -85,B 0,C 180,E1 16049.348,E2 16049.348} C_VEL
LIN {X 0,Y 267.758,Z 689.553,A -85,B 0,C 180,E1 16044.661,E2 16044.661} C_VEL
LIN {X 0,Y 266.29,Z 685.03,A -85,B 0,C 180,E1 16043.554,E2 16043.554} C_VEL
LIN {X 0,Y 266.763,Z 685.03,A -85,B 0,C 180,E1 16035.928,E2 16035.928} C_VEL
LIN {X 0,Y 267.451,Z 685.03,A -85,B 0,C 180,E1 16026.486,E2 16026.486} C_VEL
LIN {X 0,Y 268.114,Z 685.03,A -85,B 0,C 180,E1 16020.007,E2 16020.007} C_VEL
LIN {X 0,Y 267.414,Z 685.03,A -85,B 0,C 180,E1 16013.022,E2 16013.022} C_VEL
LIN {X 0,Y 266.862,Z 685.03,A -85,B 0,C 180,E1 16003.997,E2 16003.997} C_VEL
LIN {X 0,Y 266.062,Z 685.03,A -85,B 0,C 180,E1 15995.151,E2 15995.151} C_VEL
LIN {X 0,Y 265.728,Z 685.03,A -85,B 0,C 180,E1 15988.405,E2 15988.405} C_VEL
LIN {X 0,Y 265.623,Z 685.304,A -85,B 0,C 180,E1 15984.29,E2 15984.29} C_VEL
LIN {X 0,Y 267.851,Z 690.541,A -85,B 0,C 180,E1 15983.37,E2 15983.37} C_VEL
LIN {X 0,Y 270.526,Z 694.158,A -85,B 0,C 180,E1 15982.428,E2 15982.428} C_VEL
LIN {X 0,Y 286.043,Z 718.162,A -85,B 0,C 180,E1 15977.519,E2 15977.519} C_VEL
LIN {X 0,Y 298.961,Z 744.292,A -85,B 0,C 180,E1 15973.498,E2 15973.498} C_VEL
LIN {X 0,Y 306.8,Z 770.275,A -85,B 0,C 180,E1 15969.819,E2 15969.819} C_VEL
LIN {X 0,Y 307.774,Z 779.758,A -85,B 0,C 180,E1 15968.602,E2 15968.602} C_VEL
LIN {X 0,Y 301.148,Z 809.672,A -85,B 0,C 180,E1 15965.404,E2 15965.404} C_VEL
LIN {X 0,Y 293.432,Z 836.303,A -85,B 0,C 180,E1 15961.187,E2 15961.187} C_VEL
LIN {X 0,Y 285.598,Z 859.135,A -85,B 0,C 180,E1 15955.869,E2 15955.869} C_VEL
LIN {X 0,Y 278.942,Z 876.631,A -85,B 0,C 180,E1 15949.758,E2 15949.758} C_VEL
LIN {X 0,Y 274.232,Z 889.24,A -85,B 0,C 180,E1 15942.711,E2 15942.711} C_VEL
LIN {X 0,Y 272.01,Z 895.461,A -85,B 0,C 180,E1 15936.366,E2 15936.366} C_VEL
LIN {X 0,Y 271.509,Z 897.495,A -85,B 0,C 180,E1 15929.995,E2 15929.995} C_VEL
LIN {X 0,Y 272.416,Z 894.423,A -85,B 0,C 180,E1 15922.035,E2 15922.035} C_VEL
LIN {X 0,Y 275.42,Z 885.927,A -85,B 0,C 180,E1 15914.909,E2 15914.909} C_VEL
LIN {X 0,Y 280.641,Z 872.157,A -85,B 0,C 180,E1 15908.299,E2 15908.299} C_VEL
LIN {X 0,Y 287.674,Z 853.46,A -85,B 0,C 180,E1 15902.486,E2 15902.486} C_VEL
LIN {X 0,Y 295.722,Z 829.326,A -85,B 0,C 180,E1 15897.437,E2 15897.437} C_VEL
LIN {X 0,Y 303.119,Z 801.977,A -85,B 0,C 180,E1 15893.531,E2 15893.531} C_VEL
LIN {X 0,Y 308.072,Z 776.35,A -85,B 0,C 180,E1 15890.935,E2 15890.935} C_VEL
LIN {X 0,Y 301.242,Z 750.134,A -85,B 0,C 180,E1 15887.222,E2 15887.222} C_VEL
LIN {X 0,Y 288.935,Z 723.024,A -85,B 0,C 180,E1 15883.169,E2 15883.169} C_VEL
LIN {X 0,Y 272.858,Z 697.408,A -85,B 0,C 180,E1 15878.216,E2 15878.216} C_VEL
LIN {X 0,Y 267.66,Z 690.176,A -85,B 0,C 180,E1 15876.399,E2 15876.399} C_VEL
LIN {X 0,Y 268.193,Z 692.264,A -85,B 0,C 180,E1 15875.987,E2 15875.987} C_VEL
LIN {X 0,Y 284.883,Z 736.044,A -85,B 0,C 180,E1 15871.579,E2 15871.579} C_VEL
LIN {X 0,Y 289.791,Z 753.638,A -85,B 0,C 180,E1 15870.176,E2 15870.176} C_VEL
LIN {X 0,Y 286.974,Z 789.75,A -85,B 0,C 180,E1 15868.128,E2 15868.128} C_VEL
LIN {X 0,Y 283.358,Z 819.626,A -85,B 0,C 180,E1 15865.206,E2 15865.206} C_VEL
LIN {X 0,Y 279.292,Z 846.671,A -85,B 0,C 180,E1 15861.172,E2 15861.172} C_VEL
LIN {X 0,Y 275.553,Z 869.42,A -85,B 0,C 180,E1 15856.163,E2 15856.163} C_VEL
LIN {X 0,Y 272.996,Z 887.253,A -85,B 0,C 180,E1 15850.341,E2 15850.341} C_VEL
LIN {X 0,Y 272.162,Z 898.289,A -85,B 0,C 180,E1 15844.762,E2 15844.762} C_VEL
LIN {X 0,Y 272.735,Z 905.249,A -85,B 0,C 180,E1 15838.408,E2 15838.408} C_VEL
LIN {X 0,Y 274.305,Z 906.846,A -85,B 0,C 180,E1 15833.677,E2 15833.677} C_VEL
LIN {X 0,Y 278.191,Z 904.497,A -85,B 0,C 180,E1 15827.463,E2 15827.463} C_VEL
LIN {X 0,Y 284.686,Z 896.871,A -85,B 0,C 180,E1 15821.45,E2 15821.45} C_VEL
LIN {X 0,Y 294.683,Z 882.688,A -85,B 0,C 180,E1 15815.409,E2 15815.409} C_VEL
LIN {X 0,Y 307.304,Z 862.983,A -85,B 0,C 180,E1 15810.13,E2 15810.13} C_VEL
LIN {X 0,Y 323.774,Z 837.201,A -85,B 0,C 180,E1 15805.579,E2 15805.579} C_VEL
LIN {X 0,Y 336.53,Z 818.442,A -85,B 0,C 180,E1 15803.254,E2 15803.254} C_VEL
LIN {X 0,Y 334.588,Z 822.235,A -85,B 0,C 180,E1 15802.693,E2 15802.693} C_VEL
LIN {X 0,Y 330.276,Z 830.129,A -85,B 0,C 180,E1 15801.874,E2 15801.874} C_VEL
LIN {X 0,Y 321.246,Z 844.445,A -85,B 0,C 180,E1 15800.972,E2 15800.972} C_VEL
LIN {X 0,Y 313.106,Z 856.362,A -85,B 0,C 180,E1 15800.112,E2 15800.112} C_VEL
LIN {X 0,Y 312.133,Z 857.934,A -85,B 0,C 180,E1 15799.905,E2 15799.905} C_VEL
LIN {X 0,Y 289.576,Z 899.064,A -85,B 0,C 180,E1 15792.653,E2 15792.653} C_VEL
LIN {X 0,Y 275.08,Z 931.035,A -85,B 0,C 180,E1 15784.624,E2 15784.624} C_VEL
LIN {X 0,Y 266.574,Z 955.105,A -85,B 0,C 180,E1 15776.203,E2 15776.203} C_VEL
LIN {X 0,Y 262.74,Z 971.757,A -85,B 0,C 180,E1 15767.882,E2 15767.882} C_VEL
LIN {X 0,Y 261.763,Z 981.79,A -85,B 0,C 180,E1 15759.965,E2 15759.965} C_VEL
LIN {X 0,Y 261.858,Z 985.899,A -85,B 0,C 180,E1 15753.309,E2 15753.309} C_VEL
LIN {X 0,Y 262.12,Z 986.421,A -85,B 0,C 180,E1 15750.005,E2 15750.005} C_VEL
LIN {X 0,Y 261.862,Z 984.098,A -85,B 0,C 180,E1 15743.387,E2 15743.387} C_VEL
LIN {X 0,Y 262.08,Z 976.221,A -85,B 0,C 180,E1 15735.84,E2 15735.84} C_VEL
LIN {X 0,Y 264.182,Z 962.457,A -85,B 0,C 180,E1 15728.21,E2 15728.21} C_VEL
LIN {X 0,Y 269.119,Z 942.15,A -85,B 0,C 180,E1 15720.655,E2 15720.655} C_VEL
LIN {X 0,Y 276.736,Z 916.288,A -85,B 0,C 180,E1 15713.881,E2 15713.881} C_VEL
LIN {X 0,Y 286.582,Z 884.24,A -85,B 0,C 180,E1 15707.923,E2 15707.923} C_VEL
LIN {X 0,Y 297.122,Z 847.834,A -85,B 0,C 180,E1 15703.137,E2 15703.137} C_VEL
LIN {X 0,Y 307.213,Z 808.45,A -85,B 0,C 180,E1 15699.53,E2 15699.53} C_VEL
LIN {X 0,Y 308.209,Z 801.407,A -85,B 0,C 180,E1 15698.946,E2 15698.946} C_VEL
LIN {X 0,Y 293.773,Z 762.392,A -85,B 0,C 180,E1 15693.743,E2 15693.743} C_VEL
LIN {X 0,Y 274.619,Z 720.179,A -85,B 0,C 180,E1 15687.947,E2 15687.947} C_VEL
LIN {X 0,Y 258.91,Z 687.96,A -85,B 0,C 180,E1 15682.793,E2 15682.793} C_VEL
LIN {X 0,Y 258.347,Z 685.03,A -85,B 0,C 180,E1 15681.947,E2 15681.947} C_VEL
LIN {X 0,Y 258.965,Z 685.03,A -85,B 0,C 180,E1 15673.485,E2 15673.485} C_VEL
LIN {X 0,Y 259.504,Z 685.03,A -85,B 0,C 180,E1 15666.685,E2 15666.685} C_VEL
LIN {X 0,Y 260.206,Z 685.03,A -85,B 0,C 180,E1 15660.007,E2 15660.007} C_VEL
LIN {X 0,Y 259.373,Z 685.03,A -85,B 0,C 180,E1 15651.495,E2 15651.495} C_VEL
LIN {X 0,Y 258.768,Z 685.03,A -85,B 0,C 180,E1 15643.057,E2 15643.057} C_VEL
LIN {X 0,Y 258.233,Z 685.03,A -85,B 0,C 180,E1 15635.865,E2 15635.865} C_VEL
LIN {X 0,Y 257.741,Z 685.501,A -85,B 0,C 180,E1 15626.9,E2 15626.9} C_VEL
LIN {X 0,Y 260.167,Z 690.729,A -85,B 0,C 180,E1 15625.797,E2 15625.797} C_VEL
LIN {X 0,Y 262.722,Z 694.108,A -85,B 0,C 180,E1 15624.793,E2 15624.793} C_VEL
LIN {X 0,Y 277.28,Z 715.95,A -85,B 0,C 180,E1 15619.701,E2 15619.701} C_VEL
LIN {X 0,Y 291.166,Z 742.445,A -85,B 0,C 180,E1 15615.224,E2 15615.224} C_VEL
LIN {X 0,Y 299.526,Z 767.605,A -85,B 0,C 180,E1 15611.437,E2 15611.437} C_VEL
LIN {X 0,Y 301.629,Z 781.498,A -85,B 0,C 180,E1 15609.482,E2 15609.482} C_VEL
LIN {X 0,Y 294.83,Z 810.909,A -85,B 0,C 180,E1 15606.281,E2 15606.281} C_VEL
LIN {X 0,Y 286.969,Z 837.01,A -85,B 0,C 180,E1 15602.102,E2 15602.102} C_VEL
LIN {X 0,Y 278.828,Z 859.76,A -85,B 0,C 180,E1 15596.742,E2 15596.742} C_VEL
LIN {X 0,Y 271.589,Z 877.883,A -85,B 0,C 180,E1 15590.316,E2 15590.316} C_VEL
LIN {X 0,Y 266.606,Z 890.491,A -85,B 0,C 180,E1 15583.081,E2 15583.081} C_VEL
LIN {X 0,Y 264.257,Z 896.709,A -85,B 0,C 180,E1 15576.553,E2 15576.553} C_VEL
LIN {X 0,Y 263.725,Z 898.74,A -85,B 0,C 180,E1 15569.995,E2 15569.995} C_VEL
LIN {X 0,Y 264.686,Z 895.671,A -85,B 0,C 180,E1 15561.8,E2 15561.8} C_VEL
LIN {X 0,Y 267.87,Z 887.176,A -85,B 0,C 180,E1 15554.474,E2 15554.474} C_VEL
LIN {X 0,Y 273.395,Z 873.402,A -85,B 0,C 180,E1 15547.693,E2 15547.693} C_VEL
LIN {X 0,Y 280.971,Z 854.199,A -85,B 0,C 180,E1 15541.627,E2 15541.627} C_VEL
LIN {X 0,Y 289.276,Z 830.293,A -85,B 0,C 180,E1 15536.558,E2 15536.558} C_VEL
LIN {X 0,Y 296.879,Z 803.204,A -85,B 0,C 180,E1 15532.636,E2 15532.636} C_VEL
LIN {X 0,Y 301.768,Z 778.497,A -85,B 0,C 180,E1 15530.061,E2 15530.061} C_VEL
LIN {X 0,Y 295.069,Z 752.164,A -85,B 0,C 180,E1 15526.165,E2 15526.165} C_VEL
LIN {X 0,Y 282.855,Z 725.259,A -85,B 0,C 180,E1 15521.878,E2 15521.878} C_VEL
LIN {X 0,Y 267.806,Z 701.601,A -85,B 0,C 180,E1 15516.958,E2 15516.958} C_VEL
LIN {X 0,Y 264.446,Z 701.974,A -85,B 0,C 180,E1 15515.892,E2 15515.892} C_VEL
LIN {X 0,Y 281.128,Z 748.457,A -85,B 0,C 180,E1 15511.291,E2 15511.291} C_VEL
LIN {X 0,Y 282.485,Z 756.117,A -85,B 0,C 180,E1 15510.736,E2 15510.736} C_VEL
LIN {X 0,Y 279.544,Z 791.808,A -85,B 0,C 180,E1 15508.615,E2 15508.615} C_VEL
LIN {X 0,Y 275.725,Z 821.653,A -85,B 0,C 180,E1 15505.562,E2 15505.562} C_VEL
LIN {X 0,Y 271.524,Z 848.562,A -85,B 0,C 180,E1 15501.38,E2 15501.38} C_VEL
LIN {X 0,Y 267.787,Z 870.715,A -85,B 0,C 180,E1 15496.356,E2 15496.356} C_VEL
LIN {X 0,Y 265.25,Z 887.872,A -85,B 0,C 180,E1 15490.646,E2 15490.646} C_VEL
LIN {X 0,Y 264.343,Z 900.504,A -85,B 0,C 180,E1 15484.084,E2 15484.084} C_VEL
LIN {X 0,Y 264.98,Z 906.577,A -85,B 0,C 180,E1 15478.361,E2 15478.361} C_VEL
LIN {X 0,Y 266.619,Z 908.46,A -85,B 0,C 180,E1 15473.494,E2 15473.494} C_VEL
LIN {X 0,Y 270.754,Z 906.538,A -85,B 0,C 180,E1 15467.112,E2 15467.112} C_VEL
LIN {X 0,Y 278.694,Z 898.271,A -85,B 0,C 180,E1 15460.214,E2 15460.214} C_VEL
LIN {X 0,Y 290.405,Z 883.185,A -85,B 0,C 180,E1 15453.784,E2 15453.784} C_VEL
LIN {X 0,Y 305.215,Z 862.512,A -85,B 0,C 180,E1 15448.307,E2 15448.307} C_VEL
LIN {X 0,Y 323.653,Z 837.278,A -85,B 0,C 180,E1 15443.936,E2 15443.936} C_VEL
LIN {X 0,Y 327.725,Z 831.954,A -85,B 0,C 180,E1 15443.228,E2 15443.228} C_VEL
LIN {X 0,Y 312.133,Z 857.934,A -85,B 0,C 180,E1 15439.905,E2 15439.905} C_VEL
LIN {X 0,Y 302.681,Z 871.154,A -85,B 0,C 180,E1 15438.607,E2 15438.607} C_VEL
LIN {X 0,Y 294.344,Z 882.116,A -85,B 0,C 180,E1 15437.372,E2 15437.372} C_VEL
LIN {X 0,Y 293.423,Z 883.559,A -85,B 0,C 180,E1 15437.113,E2 15437.113} C_VEL
LIN {X 0,Y 274.277,Z 918.233,A -85,B 0,C 180,E1 15429.251,E2 15429.251} C_VEL
LIN {X 0,Y 261.94,Z 946.462,A -85,B 0,C 180,E1 15420.211,E2 15420.211} C_VEL
LIN {X 0,Y 256.042,Z 965.294,A -85,B 0,C 180,E1 15411.62,E2 15411.62} C_VEL
LIN {X 0,Y 254.04,Z 977.02,A -85,B 0,C 180,E1 15403.751,E2 15403.751} C_VEL
LIN {X 0,Y 253.957,Z 983.116,A -85,B 0,C 180,E1 15396.831,E2 15396.831} C_VEL
LIN {X 0,Y 254.356,Z 985.081,A -85,B 0,C 180,E1 15390.005,E2 15390.005} C_VEL
LIN {X 0,Y 254.063,Z 982.608,A -85,B 0,C 180,E1 15383.183,E2 15383.183} C_VEL
LIN {X 0,Y 254.306,Z 974.516,A -85,B 0,C 180,E1 15375.398,E2 15375.398} C_VEL
LIN {X 0,Y 256.607,Z 960.409,A -85,B 0,C 180,E1 15367.532,E2 15367.532} C_VEL
LIN {X 0,Y 261.801,Z 939.893,A -85,B 0,C 180,E1 15359.842,E2 15359.842} C_VEL
LIN {X 0,Y 270.069,Z 912.99,A -85,B 0,C 180,E1 15352.793,E2 15352.793} C_VEL
LIN {X 0,Y 280.169,Z 881.083,A -85,B 0,C 180,E1 15346.877,E2 15346.877} C_VEL
LIN {X 0,Y 290.853,Z 844.813,A -85,B 0,C 180,E1 15342.128,E2 15342.128} C_VEL
LIN {X 0,Y 301.186,Z 805.31,A -85,B 0,C 180,E1 15338.521,E2 15338.521} C_VEL
LIN {X 0,Y 290.155,Z 773.018,A -85,B 0,C 180,E1 15334.109,E2 15334.109} C_VEL
LIN {X 0,Y 273.133,Z 733.249,A -85,B 0,C 180,E1 15328.5,E2 15328.5} C_VEL
LIN {X 0,Y 250.842,Z 687.406,A -85,B 0,C 180,E1 15321.165,E2 15321.165} C_VEL
LIN {X 0,Y 250.542,Z 685.03,A -85,B 0,C 180,E1 15320.499,E2 15320.499} C_VEL
LIN {X 0,Y 250.969,Z 685.03,A -85,B 0,C 180,E1 15313.923,E2 15313.923} C_VEL
LIN {X 0,Y 251.572,Z 685.03,A -85,B 0,C 180,E1 15306.897,E2 15306.897} C_VEL
LIN {X 0,Y 252.296,Z 685.03,A -85,B 0,C 180,E1 15300.008,E2 15300.008} C_VEL
LIN {X 0,Y 251.653,Z 685.03,A -85,B 0,C 180,E1 15293.12,E2 15293.12} C_VEL
LIN {X 0,Y 250.872,Z 685.03,A -85,B 0,C 180,E1 15284.231,E2 15284.231} C_VEL
LIN {X 0,Y 250.169,Z 685.03,A -85,B 0,C 180,E1 15275.035,E2 15275.035} C_VEL
LIN {X 0,Y 249.877,Z 685.572,A -85,B 0,C 180,E1 15269.901,E2 15269.901} C_VEL
LIN {X 0,Y 252.382,Z 690.805,A -85,B 0,C 180,E1 15268.604,E2 15268.604} C_VEL
LIN {X 0,Y 254.834,Z 693.69,A -85,B 0,C 180,E1 15267.522,E2 15267.522} C_VEL
LIN {X 0,Y 270.201,Z 716.587,A -85,B 0,C 180,E1 15261.548,E2 15261.548} C_VEL
LIN {X 0,Y 283.705,Z 741.521,A -85,B 0,C 180,E1 15256.924,E2 15256.924} C_VEL
LIN {X 0,Y 292.513,Z 766.486,A -85,B 0,C 180,E1 15252.926,E2 15252.926} C_VEL
LIN {X 0,Y 295.354,Z 784.257,A -85,B 0,C 180,E1 15250.31,E2 15250.31} C_VEL
LIN {X 0,Y 288.233,Z 813.469,A -85,B 0,C 180,E1 15247.014,E2 15247.014} C_VEL
LIN {X 0,Y 279.832,Z 839.816,A -85,B 0,C 180,E1 15242.629,E2 15242.629} C_VEL
LIN {X 0,Y 271.615,Z 861.684,A -85,B 0,C 180,E1 15237.289,E2 15237.289} C_VEL
LIN {X 0,Y 264.267,Z 879.133,A -85,B 0,C 180,E1 15230.905,E2 15230.905} C_VEL
LIN {X 0,Y 259.001,Z 891.741,A -85,B 0,C 180,E1 15223.472,E2 15223.472} C_VEL
LIN {X 0,Y 256.522,Z 897.955,A -85,B 0,C 180,E1 15216.752,E2 15216.752} C_VEL
LIN {X 0,Y 255.936,Z 899.986,A -85,B 0,C 180,E1 15209.995,E2 15209.995} C_VEL
LIN {X 0,Y 256.488,Z 898.032,A -85,B 0,C 180,E1 15203.237,E2 15203.237} C_VEL
LIN {X 0,Y 259.421,Z 890.814,A -85,B 0,C 180,E1 15195.681,E2 15195.681} C_VEL
LIN {X 0,Y 264.217,Z 879.364,A -85,B 0,C 180,E1 15189.08,E2 15189.08} C_VEL
LIN {X 0,Y 271.648,Z 861.688,A -85,B 0,C 180,E1 15182.592,E2 15182.592} C_VEL
LIN {X 0,Y 280.282,Z 838.822,A -85,B 0,C 180,E1 15177.056,E2 15177.056} C_VEL
LIN {X 0,Y 288.478,Z 812.79,A -85,B 0,C 180,E1 15172.776,E2 15172.776} C_VEL
LIN {X 0,Y 295.722,Z 782.798,A -85,B 0,C 180,E1 15169.45,E2 15169.45} C_VEL
LIN {X 0,Y 290.137,Z 758.041,A -85,B 0,C 180,E1 15165.64,E2 15165.64} C_VEL
LIN {X 0,Y 279.546,Z 732.559,A -85,B 0,C 180,E1 15161.433,E2 15161.433} C_VEL
LIN {X 0,Y 266.671,Z 710.839,A -85,B 0,C 180,E1 15157.037,E2 15157.037} C_VEL
LIN {X 0,Y 261.842,Z 714.162,A -85,B 0,C 180,E1 15155.717,E2 15155.717} C_VEL
LIN {X 0,Y 262.884,Z 718.064,A -85,B 0,C 180,E1 15155.107,E2 15155.107} C_VEL
LIN {X 0,Y 275.432,Z 755.756,A -85,B 0,C 180,E1 15151.463,E2 15151.463} C_VEL
LIN {X 0,Y 272.37,Z 791.166,A -85,B 0,C 180,E1 15149.327,E2 15149.327} C_VEL
LIN {X 0,Y 268.534,Z 820.865,A -85,B 0,C 180,E1 15146.289,E2 15146.289} C_VEL
LIN {X 0,Y 264.122,Z 848.34,A -85,B 0,C 180,E1 15142.01,E2 15142.01} C_VEL
LIN {X 0,Y 260.172,Z 870.86,A -85,B 0,C 180,E1 15136.849,E2 15136.849} C_VEL
LIN {X 0,Y 257.508,Z 888.486,A -85,B 0,C 180,E1 15130.97,E2 15130.97} C_VEL
LIN {X 0,Y 256.526,Z 901.437,A -85,B 0,C 180,E1 15124.209,E2 15124.209} C_VEL
LIN {X 0,Y 257.204,Z 907.84,A -85,B 0,C 180,E1 15118.312,E2 15118.312} C_VEL
LIN {X 0,Y 258.962,Z 910.073,A -85,B 0,C 180,E1 15113.3,E2 15113.3} C_VEL
LIN {X 0,Y 263.333,Z 908.574,A -85,B 0,C 180,E1 15106.743,E2 15106.743} C_VEL
LIN {X 0,Y 271.727,Z 900.966,A -85,B 0,C 180,E1 15099.685,E2 15099.685} C_VEL
LIN {X 0,Y 284.04,Z 886.901,A -85,B 0,C 180,E1 15093.15,E2 15093.15} C_VEL
LIN {X 0,Y 299.541,Z 867.7,A -85,B 0,C 180,E1 15087.634,E2 15087.634} C_VEL
LIN {X 0,Y 318.106,Z 845.175,A -85,B 0,C 180,E1 15083.355,E2 15083.355} C_VEL
LIN {X 0,Y 310.51,Z 856.654,A -85,B 0,C 180,E1 15081.605,E2 15081.605} C_VEL
LIN {X 0,Y 293.423,Z 883.559,A -85,B 0,C 180,E1 15077.113,E2 15077.113} C_VEL
LIN {X 0,Y 283.904,Z 895.647,A -85,B 0,C 180,E1 15075.387,E2 15075.387} C_VEL
LIN {X 0,Y 275.509,Z 905.601,A -85,B 0,C 180,E1 15073.769,E2 15073.769} C_VEL
LIN {X 0,Y 274.664,Z 906.922,A -85,B 0,C 180,E1 15073.458,E2 15073.458} C_VEL
LIN {X 0,Y 257.867,Z 938.972,A -85,B 0,C 180,E1 15063.783,E2 15063.783} C_VEL
LIN {X 0,Y 249.383,Z 961.099,A -85,B 0,C 180,E1 15054.114,E2 15054.114} C_VEL
LIN {X 0,Y 246.342,Z 974.805,A -85,B 0,C 180,E1 15045.097,E2 15045.097} C_VEL
LIN {X 0,Y 246.117,Z 981.866,A -85,B 0,C 180,E1 15037.049,E2 15037.049} C_VEL
LIN {X 0,Y 246.589,Z 983.724,A -85,B 0,C 180,E1 15030.005,E2 15030.005} C_VEL
LIN {X 0,Y 246.256,Z 981.084,A -85,B 0,C 180,E1 15022.965,E2 15022.965} C_VEL
LIN {X 0,Y 246.447,Z 973.935,A -85,B 0,C 180,E1 15015.828,E2 15015.828} C_VEL
LIN {X 0,Y 248.64,Z 960.176,A -85,B 0,C 180,E1 15007.713,E2 15007.713} C_VEL
LIN {X 0,Y 253.462,Z 941.442,A -85,B 0,C 180,E1 15000.269,E2 15000.269} C_VEL
LIN {X 0,Y 261.272,Z 916.286,A -85,B 0,C 180,E1 14993.19,E2 14993.19} C_VEL
LIN {X 0,Y 271.216,Z 885.714,A -85,B 0,C 180,E1 14987.063,E2 14987.063} C_VEL
LIN {X 0,Y 282.598,Z 849.045,A -85,B 0,C 180,E1 14981.911,E2 14981.911} C_VEL
LIN {X 0,Y 293.414,Z 809.354,A -85,B 0,C 180,E1 14978.054,E2 14978.054} C_VEL
LIN {X 0,Y 293.32,Z 803.677,A -85,B 0,C 180,E1 14977.428,E2 14977.428} C_VEL
LIN {X 0,Y 279.493,Z 765.835,A -85,B 0,C 180,E1 14971.996,E2 14971.996} C_VEL
LIN {X 0,Y 261.872,Z 725.971,A -85,B 0,C 180,E1 14966.07,E2 14966.07} C_VEL
LIN {X 0,Y 242.64,Z 685.477,A -85,B 0,C 180,E1 14959.181,E2 14959.181} C_VEL
LIN {X 0,Y 243.323,Z 685.03,A -85,B 0,C 180,E1 14950.729,E2 14950.729} C_VEL
LIN {X 0,Y 244.048,Z 685.03,A -85,B 0,C 180,E1 14943.553,E2 14943.553} C_VEL
LIN {X 0,Y 244.386,Z 685.03,A -85,B 0,C 180,E1 14940.008,E2 14940.008} C_VEL
LIN {X 0,Y 243.616,Z 685.03,A -85,B 0,C 180,E1 14932.318,E2 14932.318} C_VEL
LIN {X 0,Y 243.098,Z 685.03,A -85,B 0,C 180,E1 14925.633,E2 14925.633} C_VEL
LIN {X 0,Y 242.434,Z 685.03,A -85,B 0,C 180,E1 14918.081,E2 14918.081} C_VEL
LIN {X 0,Y 242.098,Z 685.726,A -85,B 0,C 180,E1 14913.396,E2 14913.396} C_VEL
LIN {X 0,Y 244.389,Z 690.675,A -85,B 0,C 180,E1 14911.981,E2 14911.981} C_VEL
LIN {X 0,Y 247.305,Z 693.957,A -85,B 0,C 180,E1 14910.487,E2 14910.487} C_VEL
LIN {X 0,Y 257.655,Z 709.141,A -85,B 0,C 180,E1 14905.732,E2 14905.732} C_VEL
LIN {X 0,Y 270.581,Z 729.565,A -85,B 0,C 180,E1 14900.884,E2 14900.884} C_VEL
LIN {X 0,Y 281.862,Z 753.842,A -85,B 0,C 180,E1 14896.44,E2 14896.44} C_VEL
LIN {X 0,Y 288.516,Z 778.591,A -85,B 0,C 180,E1 14892.389,E2 14892.389} C_VEL
LIN {X 0,Y 288.963,Z 787.613,A -85,B 0,C 180,E1 14891.107,E2 14891.107} C_VEL
LIN {X 0,Y 281.294,Z 817.353,A -85,B 0,C 180,E1 14887.601,E2 14887.601} C_VEL
LIN {X 0,Y 272.666,Z 842.873,A -85,B 0,C 180,E1 14883.124,E2 14883.124} C_VEL
LIN {X 0,Y 264.132,Z 864.21,A -85,B 0,C 180,E1 14877.66,E2 14877.66} C_VEL
LIN {X 0,Y 256.982,Z 880.383,A -85,B 0,C 180,E1 14871.526,E2 14871.526} C_VEL
LIN {X 0,Y 251.401,Z 892.992,A -85,B 0,C 180,E1 14863.887,E2 14863.887} C_VEL
LIN {X 0,Y 248.774,Z 899.203,A -85,B 0,C 180,E1 14856.963,E2 14856.963} C_VEL
LIN {X 0,Y 248.152,Z 901.231,A -85,B 0,C 180,E1 14849.995,E2 14849.995} C_VEL
LIN {X 0,Y 249.261,Z 898.163,A -85,B 0,C 180,E1 14841.289,E2 14841.289} C_VEL
LIN {X 0,Y 252.831,Z 889.674,A -85,B 0,C 180,E1 14833.524,E2 14833.524} C_VEL
LIN {X 0,Y 259.014,Z 875.89,A -85,B 0,C 180,E1 14826.382,E2 14826.382} C_VEL
LIN {X 0,Y 267.467,Z 856.332,A -85,B 0,C 180,E1 14819.945,E2 14819.945} C_VEL
LIN {X 0,Y 276.153,Z 833.46,A -85,B 0,C 180,E1 14814.909,E2 14814.909} C_VEL
LIN {X 0,Y 284.644,Z 805.653,A -85,B 0,C 180,E1 14810.731,E2 14810.731} C_VEL
LIN {X 0,Y 289.394,Z 783.323,A -85,B 0,C 180,E1 14808.269,E2 14808.269} C_VEL
LIN {X 0,Y 283.65,Z 758.767,A -85,B 0,C 180,E1 14804.283,E2 14804.283} C_VEL
LIN {X 0,Y 273.287,Z 734.396,A -85,B 0,C 180,E1 14799.947,E2 14799.947} C_VEL
LIN {X 0,Y 264.851,Z 720.727,A -85,B 0,C 180,E1 14796.943,E2 14796.943} C_VEL
LIN {X 0,Y 259.438,Z 726.807,A -85,B 0,C 180,E1 14795.553,E2 14795.553} C_VEL
LIN {X 0,Y 258.504,Z 727.378,A -85,B 0,C 180,E1 14795.077,E2 14795.077} C_VEL
LIN {X 0,Y 268.197,Z 757.349,A -85,B 0,C 180,E1 14792.114,E2 14792.114} C_VEL
LIN {X 0,Y 264.832,Z 794.042,A -85,B 0,C 180,E1 14789.777,E2 14789.777} C_VEL
LIN {X 0,Y 260.601,Z 824.992,A -85,B 0,C 180,E1 14786.394,E2 14786.394} C_VEL
LIN {X 0,Y 255.965,Z 852.177,A -85,B 0,C 180,E1 14781.838,E2 14781.838} C_VEL
LIN {X 0,Y 251.997,Z 874.531,A -85,B 0,C 180,E1 14776.362,E2 14776.362} C_VEL
LIN {X 0,Y 249.515,Z 891.003,A -85,B 0,C 180,E1 14770.444,E2 14770.444} C_VEL
LIN {X 0,Y 248.729,Z 903.602,A -85,B 0,C 180,E1 14763.47,E2 14763.47} C_VEL
LIN {X 0,Y 249.799,Z 910.282,A -85,B 0,C 180,E1 14756.529,E2 14756.529} C_VEL
LIN {X 0,Y 253.189,Z 911.78,A -85,B 0,C 180,E1 14749.693,E2 14749.693} C_VEL
LIN {X 0,Y 259.347,Z 908.311,A -85,B 0,C 180,E1 14743.081,E2 14743.081} C_VEL
LIN {X 0,Y 270.031,Z 898.677,A -85,B 0,C 180,E1 14736.094,E2 14736.094} C_VEL
LIN {X 0,Y 285.706,Z 881.949,A -85,B 0,C 180,E1 14729.44,E2 14729.44} C_VEL
LIN {X 0,Y 306.914,Z 858.743,A -85,B 0,C 180,E1 14723.839,E2 14723.839} C_VEL
LIN {X 0,Y 308.977,Z 856.522,A -85,B 0,C 180,E1 14723.441,E2 14723.441} C_VEL
LIN {X 0,Y 302.287,Z 865.664,A -85,B 0,C 180,E1 14721.846,E2 14721.846} C_VEL
LIN {X 0,Y 276.304,Z 904.16,A -85,B 0,C 180,E1 14714.142,E2 14714.142} C_VEL
LIN {X 0,Y 274.664,Z 906.922,A -85,B 0,C 180,E1 14713.458,E2 14713.458} C_VEL
LIN {X 0,Y 265.571,Z 917.711,A -85,B 0,C 180,E1 14711.224,E2 14711.224} C_VEL
LIN {X 0,Y 256.807,Z 927.735,A -85,B 0,C 180,E1 14708.746,E2 14708.746} C_VEL
LIN {X 0,Y 244.418,Z 953.136,A -85,B 0,C 180,E1 14698.593,E2 14698.593} C_VEL
LIN {X 0,Y 239.324,Z 969.53,A -85,B 0,C 180,E1 14688.942,E2 14688.942} C_VEL
LIN {X 0,Y 238.225,Z 978.145,A -85,B 0,C 180,E1 14680.961,E2 14680.961} C_VEL
LIN {X 0,Y 238.441,Z 981.999,A -85,B 0,C 180,E1 14673.634,E2 14673.634} C_VEL
LIN {X 0,Y 238.805,Z 982.347,A -85,B 0,C 180,E1 14670.006,E2 14670.006} C_VEL
LIN {X 0,Y 238.476,Z 979.533,A -85,B 0,C 180,E1 14662.735,E2 14662.735} C_VEL
LIN {X 0,Y 238.685,Z 972.134,A -85,B 0,C 180,E1 14655.357,E2 14655.357} C_VEL
LIN {X 0,Y 241.088,Z 958.039,A -85,B 0,C 180,E1 14646.997,E2 14646.997} C_VEL
LIN {X 0,Y 246.57,Z 937.772,A -85,B 0,C 180,E1 14638.966,E2 14638.966} C_VEL
LIN {X 0,Y 255.219,Z 911.172,A -85,B 0,C 180,E1 14631.628,E2 14631.628} C_VEL
LIN {X 0,Y 265.99,Z 879,A -85,B 0,C 180,E1 14625.392,E2 14625.392} C_VEL
LIN {X 0,Y 277.483,Z 842.218,A -85,B 0,C 180,E1 14620.421,E2 14620.421} C_VEL
LIN {X 0,Y 286.723,Z 807.659,A -85,B 0,C 180,E1 14617.075,E2 14617.075} C_VEL
LIN {X 0,Y 273.217,Z 769.75,A -85,B 0,C 180,E1 14611.421,E2 14611.421} C_VEL
LIN {X 0,Y 255.766,Z 729.344,A -85,B 0,C 180,E1 14605.192,E2 14605.192} C_VEL
LIN {X 0,Y 234.793,Z 685.03,A -85,B 0,C 180,E1 14597.343,E2 14597.343} C_VEL
LIN {X 0,Y 235.337,Z 685.03,A -85,B 0,C 180,E1 14591.098,E2 14591.098} C_VEL
LIN {X 0,Y 236.106,Z 685.03,A -85,B 0,C 180,E1 14583.672,E2 14583.672} C_VEL
LIN {X 0,Y 236.483,Z 685.03,A -85,B 0,C 180,E1 14580.008,E2 14580.008} C_VEL
LIN {X 0,Y 235.772,Z 685.03,A -85,B 0,C 180,E1 14572.655,E2 14572.655} C_VEL
LIN {X 0,Y 234.98,Z 685.03,A -85,B 0,C 180,E1 14564.414,E2 14564.414} C_VEL
LIN {X 0,Y 234.448,Z 685.066,A -85,B 0,C 180,E1 14557.688,E2 14557.688} C_VEL
LIN {X 0,Y 236.096,Z 690.085,A -85,B 0,C 180,E1 14556.293,E2 14556.293} C_VEL
LIN {X 0,Y 239.631,Z 693.563,A -85,B 0,C 180,E1 14554.105,E2 14554.105} C_VEL
LIN {X 0,Y 249.736,Z 708.365,A -85,B 0,C 180,E1 14548.66,E2 14548.66} C_VEL
LIN {X 0,Y 263.235,Z 729.243,A -85,B 0,C 180,E1 14542.994,E2 14542.994} C_VEL
LIN {X 0,Y 274.302,Z 751.815,A -85,B 0,C 180,E1 14538.44,E2 14538.44} C_VEL
LIN {X 0,Y 281.305,Z 774.734,A -85,B 0,C 180,E1 14534.412,E2 14534.412} C_VEL
LIN {X 0,Y 283.434,Z 787.728,A -85,B 0,C 180,E1 14532.246,E2 14532.246} C_VEL
LIN {X 0,Y 275.563,Z 817.268,A -85,B 0,C 180,E1 14528.776,E2 14528.776} C_VEL
LIN {X 0,Y 266.812,Z 842.306,A -85,B 0,C 180,E1 14524.438,E2 14524.438} C_VEL
LIN {X 0,Y 257.695,Z 864.476,A -85,B 0,C 180,E1 14518.787,E2 14518.787} C_VEL
LIN {X 0,Y 249.727,Z 881.632,A -85,B 0,C 180,E1 14512.185,E2 14512.185} C_VEL
LIN {X 0,Y 243.832,Z 894.24,A -85,B 0,C 180,E1 14504.328,E2 14504.328} C_VEL
LIN {X 0,Y 241.025,Z 900.452,A -85,B 0,C 180,E1 14497.188,E2 14497.188} C_VEL
LIN {X 0,Y 240.364,Z 902.476,A -85,B 0,C 180,E1 14489.995,E2 14489.995} C_VEL
LIN {X 0,Y 241.57,Z 899.407,A -85,B 0,C 180,E1 14481.01,E2 14481.01} C_VEL
LIN {X 0,Y 245.358,Z 890.919,A -85,B 0,C 180,E1 14473.008,E2 14473.008} C_VEL
LIN {X 0,Y 251.881,Z 877.134,A -85,B 0,C 180,E1 14465.67,E2 14465.67} C_VEL
LIN {X 0,Y 260.738,Z 857.574,A -85,B 0,C 180,E1 14459.087,E2 14459.087} C_VEL
LIN {X 0,Y 270.081,Z 834.03,A -85,B 0,C 180,E1 14453.835,E2 14453.835} C_VEL
LIN {X 0,Y 278.661,Z 806.876,A -85,B 0,C 180,E1 14449.718,E2 14449.718} C_VEL
LIN {X 0,Y 283.372,Z 786.154,A -85,B 0,C 180,E1 14447.382,E2 14447.382} C_VEL
LIN {X 0,Y 277.72,Z 760.967,A -85,B 0,C 180,E1 14443.098,E2 14443.098} C_VEL
LIN {X 0,Y 267.687,Z 737.014,A -85,B 0,C 180,E1 14438.567,E2 14438.567} C_VEL
LIN {X 0,Y 263.794,Z 731.321,A -85,B 0,C 180,E1 14437.116,E2 14437.116} C_VEL
LIN {X 0,Y 259.484,Z 736.144,A -85,B 0,C 180,E1 14436.067,E2 14436.067} C_VEL
LIN {X 0,Y 256.041,Z 739.583,A -85,B 0,C 180,E1 14435.156,E2 14435.156} C_VEL
LIN {X 0,Y 255.178,Z 740.26,A -85,B 0,C 180,E1 14434.666,E2 14434.666} C_VEL
LIN {X 0,Y 260.852,Z 760.789,A -85,B 0,C 180,E1 14432.689,E2 14432.689} C_VEL
LIN {X 0,Y 257.342,Z 796.838,A -85,B 0,C 180,E1 14430.248,E2 14430.248} C_VEL
LIN {X 0,Y 252.771,Z 828.078,A -85,B 0,C 180,E1 14426.614,E2 14426.614} C_VEL
LIN {X 0,Y 247.963,Z 854.921,A -85,B 0,C 180,E1 14421.875,E2 14421.875} C_VEL
LIN {X 0,Y 244.032,Z 876.651,A -85,B 0,C 180,E1 14416.258,E2 14416.258} C_VEL
LIN {X 0,Y 241.513,Z 893.526,A -85,B 0,C 180,E1 14409.885,E2 14409.885} C_VEL
LIN {X 0,Y 240.969,Z 905.675,A -85,B 0,C 180,E1 14402.684,E2 14402.684} C_VEL
LIN {X 0,Y 242.048,Z 911.609,A -85,B 0,C 180,E1 14396.418,E2 14396.418} C_VEL
LIN {X 0,Y 245.624,Z 913.55,A -85,B 0,C 180,E1 14389.372,E2 14389.372} C_VEL
LIN {X 0,Y 252.155,Z 910.647,A -85,B 0,C 180,E1 14382.583,E2 14382.583} C_VEL
LIN {X 0,Y 263.382,Z 901.791,A -85,B 0,C 180,E1 14375.451,E2 14375.451} C_VEL
LIN {X 0,Y 280.792,Z 885.346,A -85,B 0,C 180,E1 14368.396,E2 14368.396} C_VEL
LIN {X 0,Y 299.765,Z 866.885,A -85,B 0,C 180,E1 14363.525,E2 14363.525} C_VEL
LIN {X 0,Y 267.059,Z 910.955,A -85,B 0,C 180,E1 14353.813,E2 14353.813} C_VEL
LIN {X 0,Y 256.807,Z 927.735,A -85,B 0,C 180,E1 14348.746,E2 14348.746} C_VEL
LIN {X 0,Y 248.388,Z 937.09,A -85,B 0,C 180,E1 14345.953,E2 14345.953} C_VEL
LIN {X 0,Y 240.476,Z 945.585,A -85,B 0,C 180,E1 14342.884,E2 14342.884} C_VEL
LIN {X 0,Y 232.782,Z 963.915,A -85,B 0,C 180,E1 14332.896,E2 14332.896} C_VEL
LIN {X 0,Y 230.412,Z 975.329,A -85,B 0,C 180,E1 14323.258,E2 14323.258} C_VEL
LIN {X 0,Y 230.436,Z 979.282,A -85,B 0,C 180,E1 14317.532,E2 14317.532} C_VEL
LIN {X 0,Y 231.036,Z 980.925,A -85,B 0,C 180,E1 14310.006,E2 14310.006} C_VEL
LIN {X 0,Y 230.695,Z 977.929,A -85,B 0,C 180,E1 14302.488,E2 14302.488} C_VEL
LIN {X 0,Y 230.96,Z 970.234,A -85,B 0,C 180,E1 14294.855,E2 14294.855} C_VEL
LIN {X 0,Y 233.504,Z 956.176,A -85,B 0,C 180,E1 14286.415,E2 14286.415} C_VEL
LIN {X 0,Y 239.127,Z 936.164,A -85,B 0,C 180,E1 14278.339,E2 14278.339} C_VEL
LIN {X 0,Y 248.055,Z 909.577,A -85,B 0,C 180,E1 14270.87,E2 14270.87} C_VEL
LIN {X 0,Y 259.024,Z 877.617,A -85,B 0,C 180,E1 14264.569,E2 14264.569} C_VEL
LIN {X 0,Y 270.819,Z 840.962,A -85,B 0,C 180,E1 14259.543,E2 14259.543} C_VEL
LIN {X 0,Y 279.531,Z 809.752,A -85,B 0,C 180,E1 14256.433,E2 14256.433} C_VEL
LIN {X 0,Y 265.998,Z 771.201,A -85,B 0,C 180,E1 14250.471,E2 14250.471} C_VEL
LIN {X 0,Y 248.615,Z 730.79,A -85,B 0,C 180,E1 14243.971,E2 14243.971} C_VEL
LIN {X 0,Y 228.923,Z 690.311,A -85,B 0,C 180,E1 14236.685,E2 14236.685} C_VEL
LIN {X 0,Y 227.09,Z 685.03,A -85,B 0,C 180,E1 14234.437,E2 14234.437} C_VEL
LIN {X 0,Y 227.815,Z 685.03,A -85,B 0,C 180,E1 14226.525,E2 14226.525} C_VEL
LIN {X 0,Y 228.57,Z 685.03,A -85,B 0,C 180,E1 14220.008,E2 14220.008} C_VEL
LIN {X 0,Y 227.825,Z 685.03,A -85,B 0,C 180,E1 14212.397,E2 14212.397} C_VEL
LIN {X 0,Y 226.928,Z 685.449,A -85,B 0,C 180,E1 14203.223,E2 14203.223} C_VEL
LIN {X 0,Y 228.82,Z 690.261,A -85,B 0,C 180,E1 14201.133,E2 14201.133} C_VEL
LIN {X 0,Y 232.313,Z 693.58,A -85,B 0,C 180,E1 14198.338,E2 14198.338} C_VEL
LIN {X 0,Y 236.068,Z 699.141,A -85,B 0,C 180,E1 14195.619,E2 14195.619} C_VEL
LIN {X 0,Y 246.294,Z 713.869,A -85,B 0,C 180,E1 14189.735,E2 14189.735} C_VEL
LIN {X 0,Y 259.973,Z 735.895,A -85,B 0,C 180,E1 14183.632,E2 14183.632} C_VEL
LIN {X 0,Y 270.261,Z 758.605,A -85,B 0,C 180,E1 14178.881,E2 14178.881} C_VEL
LIN {X 0,Y 276.415,Z 782.599,A -85,B 0,C 180,E1 14174.527,E2 14174.527} C_VEL
LIN {X 0,Y 277.006,Z 791.739,A -85,B 0,C 180,E1 14173.056,E2 14173.056} C_VEL
LIN {X 0,Y 268.677,Z 821.062,A -85,B 0,C 180,E1 14169.443,E2 14169.443} C_VEL
LIN {X 0,Y 258.996,Z 847.187,A -85,B 0,C 180,E1 14164.612,E2 14164.612} C_VEL
LIN {X 0,Y 249.35,Z 868.937,A -85,B 0,C 180,E1 14158.571,E2 14158.571} C_VEL
LIN {X 0,Y 241.651,Z 884.635,A -85,B 0,C 180,E1 14151.999,E2 14151.999} C_VEL
LIN {X 0,Y 236.258,Z 895.492,A -85,B 0,C 180,E1 14144.797,E2 14144.797} C_VEL
LIN {X 0,Y 233.288,Z 901.7,A -85,B 0,C 180,E1 14137.428,E2 14137.428} C_VEL
LIN {X 0,Y 232.579,Z 903.721,A -85,B 0,C 180,E1 14129.994,E2 14129.994} C_VEL
LIN {X 0,Y 233.857,Z 900.656,A -85,B 0,C 180,E1 14120.71,E2 14120.71} C_VEL
LIN {X 0,Y 238.054,Z 891.878,A -85,B 0,C 180,E1 14112.249,E2 14112.249} C_VEL
LIN {X 0,Y 245.274,Z 877.362,A -85,B 0,C 180,E1 14104.483,E2 14104.483} C_VEL
LIN {X 0,Y 254.74,Z 857.297,A -85,B 0,C 180,E1 14097.775,E2 14097.775} C_VEL
LIN {X 0,Y 264.682,Z 832.96,A -85,B 0,C 180,E1 14092.42,E2 14092.42} C_VEL
LIN {X 0,Y 273.561,Z 805.422,A -85,B 0,C 180,E1 14088.325,E2 14088.325} C_VEL
LIN {X 0,Y 277.345,Z 788.622,A -85,B 0,C 180,E1 14086.396,E2 14086.396} C_VEL
LIN {X 0,Y 272.323,Z 764.636,A -85,B 0,C 180,E1 14082.116,E2 14082.116} C_VEL
LIN {X 0,Y 263.106,Z 741.706,A -85,B 0,C 180,E1 14077.532,E2 14077.532} C_VEL
LIN {X 0,Y 261.319,Z 742.582,A -85,B 0,C 180,E1 14077.052,E2 14077.052} C_VEL
LIN {X 0,Y 252.599,Z 751.699,A -85,B 0,C 180,E1 14074.928,E2 14074.928} C_VEL
LIN {X 0,Y 251.222,Z 751.942,A -85,B 0,C 180,E1 14074.373,E2 14074.373} C_VEL
LIN {X 0,Y 253.65,Z 762.346,A -85,B 0,C 180,E1 14073.396,E2 14073.396} C_VEL
LIN {X 0,Y 249.946,Z 798.069,A -85,B 0,C 180,E1 14070.863,E2 14070.863} C_VEL
LIN {X 0,Y 245.474,Z 827.964,A -85,B 0,C 180,E1 14067.312,E2 14067.312} C_VEL
LIN {X 0,Y 240.573,Z 854.482,A -85,B 0,C 180,E1 14062.583,E2 14062.583} C_VEL
LIN {X 0,Y 236.405,Z 876.917,A -85,B 0,C 180,E1 14056.741,E2 14056.741} C_VEL
LIN {X 0,Y 233.739,Z 893.994,A -85,B 0,C 180,E1 14050.217,E2 14050.217} C_VEL
LIN {X 0,Y 233.143,Z 906.625,A -85,B 0,C 180,E1 14042.774,E2 14042.774} C_VEL
LIN {X 0,Y 234.286,Z 912.934,A -85,B 0,C 180,E1 14036.299,E2 14036.299} C_VEL
LIN {X 0,Y 238.058,Z 915.305,A -85,B 0,C 180,E1 14029.03,E2 14029.03} C_VEL
LIN {X 0,Y 244.979,Z 912.98,A -85,B 0,C 180,E1 14022.055,E2 14022.055} C_VEL
LIN {X 0,Y 256.783,Z 904.952,A -85,B 0,C 180,E1 14014.777,E2 14014.777} C_VEL
LIN {X 0,Y 274.986,Z 889.761,A -85,B 0,C 180,E1 14007.648,E2 14007.648} C_VEL
LIN {X 0,Y 290.587,Z 876.258,A -85,B 0,C 180,E1 14003.617,E2 14003.617} C_VEL
LIN {X 0,Y 257.782,Z 917.082,A -85,B 0,C 180,E1 13993.491,E2 13993.491} C_VEL
LIN {X 0,Y 240.476,Z 945.585,A -85,B 0,C 180,E1 13982.884,E2 13982.884} C_VEL
LIN {X 0,Y 233.036,Z 953.222,A -85,B 0,C 180,E1 13979.497,E2 13979.497} C_VEL
LIN {X 0,Y 226.457,Z 959.889,A -85,B 0,C 180,E1 13975.805,E2 13975.805} C_VEL
LIN {X 0,Y 222.812,Z 972.388,A -85,B 0,C 180,E1 13965.725,E2 13965.725} C_VEL
LIN {X 0,Y 222.594,Z 977.966,A -85,B 0,C 180,E1 13957.799,E2 13957.799} C_VEL
LIN {X 0,Y 223.259,Z 979.453,A -85,B 0,C 180,E1 13950.006,E2 13950.006} C_VEL
LIN {X 0,Y 222.906,Z 976.241,A -85,B 0,C 180,E1 13942.224,E2 13942.224} C_VEL
LIN {X 0,Y 223.253,Z 968.268,A -85,B 0,C 180,E1 13934.319,E2 13934.319} C_VEL
LIN {X 0,Y 225.984,Z 953.923,A -85,B 0,C 180,E1 13925.66,E2 13925.66} C_VEL
LIN {X 0,Y 232.055,Z 933.404,A -85,B 0,C 180,E1 13917.327,E2 13917.327} C_VEL
LIN {X 0,Y 241.387,Z 906.619,A -85,B 0,C 180,E1 13909.767,E2 13909.767} C_VEL
LIN {X 0,Y 252.557,Z 874.762,A -85,B 0,C 180,E1 13903.48,E2 13903.48} C_VEL
LIN {X 0,Y 265.157,Z 836.767,A -85,B 0,C 180,E1 13898.31,E2 13898.31} C_VEL
LIN {X 0,Y 272.211,Z 811.553,A -85,B 0,C 180,E1 13895.746,E2 13895.746} C_VEL
LIN {X 0,Y 259.099,Z 773.688,A -85,B 0,C 180,E1 13889.678,E2 13889.678} C_VEL
LIN {X 0,Y 242.467,Z 734.268,A -85,B 0,C 180,E1 13883.089,E2 13883.089} C_VEL
LIN {X 0,Y 227.561,Z 701.799,A -85,B 0,C 180,E1 13876.999,E2 13876.999} C_VEL
LIN {X 0,Y 225.662,Z 694.685,A -85,B 0,C 180,E1 13874.651,E2 13874.651} C_VEL
LIN {X 0,Y 224.805,Z 692.585,A -85,B 0,C 180,E1 13873.596,E2 13873.596} C_VEL
LIN {X 0,Y 220.424,Z 687.964,A -85,B 0,C 180,E1 13867.311,E2 13867.311} C_VEL
LIN {X 0,Y 220.033,Z 685.03,A -85,B 0,C 180,E1 13865.075,E2 13865.075} C_VEL
LIN {X 0,Y 220.656,Z 685.03,A -85,B 0,C 180,E1 13860.009,E2 13860.009} C_VEL
LIN {X 0,Y 219.909,Z 685.541,A -85,B 0,C 180,E1 13852.243,E2 13852.243} C_VEL
LIN {X 0,Y 221.38,Z 690.104,A -85,B 0,C 180,E1 13848.708,E2 13848.708} C_VEL
LIN {X 0,Y 225.215,Z 693.613,A -85,B 0,C 180,E1 13843.841,E2 13843.841} C_VEL
LIN {X 0,Y 228.942,Z 699.312,A -85,B 0,C 180,E1 13840.156,E2 13840.156} C_VEL
LIN {X 0,Y 231.314,Z 703.203,A -85,B 0,C 180,E1 13838.166,E2 13838.166} C_VEL
LIN {X 0,Y 235.921,Z 709.56,A -85,B 0,C 180,E1 13834.926,E2 13834.926} C_VEL
LIN {X 0,Y 244.55,Z 722.231,A -85,B 0,C 180,E1 13829.973,E2 13829.973} C_VEL
LIN {X 0,Y 257.282,Z 743.821,A -85,B 0,C 180,E1 13823.973,E2 13823.973} C_VEL
LIN {X 0,Y 266.318,Z 766.534,A -85,B 0,C 180,E1 13819.123,E2 13819.123} C_VEL
LIN {X 0,Y 271.21,Z 790.195,A -85,B 0,C 180,E1 13814.669,E2 13814.669} C_VEL
LIN {X 0,Y 270.443,Z 796.628,A -85,B 0,C 180,E1 13813.809,E2 13813.809} C_VEL
LIN {X 0,Y 261.42,Z 825.915,A -85,B 0,C 180,E1 13809.95,E2 13809.95} C_VEL
LIN {X 0,Y 251.111,Z 851.816,A -85,B 0,C 180,E1 13804.808,E2 13804.808} C_VEL
LIN {X 0,Y 240.969,Z 873.236,A -85,B 0,C 180,E1 13798.355,E2 13798.355} C_VEL
LIN {X 0,Y 232.764,Z 889.107,A -85,B 0,C 180,E1 13790.884,E2 13790.884} C_VEL
LIN {X 0,Y 227.684,Z 898.708,A -85,B 0,C 180,E1 13783.408,E2 13783.408} C_VEL
LIN {X 0,Y 225.576,Z 902.945,A -85,B 0,C 180,E1 13777.683,E2 13777.683} C_VEL
LIN {X 0,Y 224.778,Z 904.969,A -85,B 0,C 180,E1 13769.994,E2 13769.994} C_VEL
LIN {X 0,Y 225.536,Z 903.019,A -85,B 0,C 180,E1 13762.304,E2 13762.304} C_VEL
LIN {X 0,Y 228.688,Z 896.867,A -85,B 0,C 180,E1 13754.689,E2 13754.689} C_VEL
LIN {X 0,Y 235.254,Z 884.353,A -85,B 0,C 180,E1 13746.358,E2 13746.358} C_VEL
LIN {X 0,Y 244.153,Z 867.017,A -85,B 0,C 180,E1 13739.335,E2 13739.335} C_VEL
LIN {X 0,Y 254.067,Z 845.206,A -85,B 0,C 180,E1 13733.554,E2 13733.554} C_VEL
LIN {X 0,Y 263.897,Z 819.027,A -85,B 0,C 180,E1 13728.875,E2 13728.875} C_VEL
LIN {X 0,Y 271.46,Z 792.046,A -85,B 0,C 180,E1 13725.55,E2 13725.55} C_VEL
LIN {X 0,Y 267.263,Z 769.455,A -85,B 0,C 180,E1 13721.339,E2 13721.339} C_VEL
LIN {X 0,Y 260.927,Z 751.472,A -85,B 0,C 180,E1 13717.638,E2 13717.638} C_VEL
LIN {X 0,Y 246.568,Z 764.655,A -85,B 0,C 180,E1 13714.165,E2 13714.165} C_VEL
LIN {X 0,Y 242.002,Z 803.609,A -85,B 0,C 180,E1 13711.077,E2 13711.077} C_VEL
LIN {X 0,Y 237.28,Z 832.937,A -85,B 0,C 180,E1 13707.25,E2 13707.25} C_VEL
LIN {X 0,Y 232.057,Z 860.063,A -85,B 0,C 180,E1 13701.946,E2 13701.946} C_VEL
LIN {X 0,Y 227.753,Z 882.711,A -85,B 0,C 180,E1 13695.358,E2 13695.358} C_VEL
LIN {X 0,Y 225.456,Z 900.111,A -85,B 0,C 180,E1 13687.684,E2 13687.684} C_VEL
LIN {X 0,Y 225.738,Z 910.823,A -85,B 0,C 180,E1 13679.991,E2 13679.991} C_VEL
LIN {X 0,Y 228.256,Z 916.219,A -85,B 0,C 180,E1 13672.394,E2 13672.394} C_VEL
LIN {X 0,Y 233.777,Z 916.706,A -85,B 0,C 180,E1 13665.03,E2 13665.03} C_VEL
LIN {X 0,Y 242.791,Z 912.72,A -85,B 0,C 180,E1 13658.098,E2 13658.098} C_VEL
LIN {X 0,Y 259.034,Z 901.808,A -85,B 0,C 180,E1 13650.313,E2 13650.313} C_VEL
LIN {X 0,Y 281.47,Z 884.845,A -85,B 0,C 180,E1 13643.542,E2 13643.542} C_VEL
LIN {X 0,Y 253.072,Z 916.73,A -85,B 0,C 180,E1 13635.157,E2 13635.157} C_VEL
LIN {X 0,Y 234.151,Z 944.315,A -85,B 0,C 180,E1 13624.422,E2 13624.422} C_VEL
LIN {X 0,Y 226.457,Z 959.889,A -85,B 0,C 180,E1 13615.805,E2 13615.805} C_VEL
LIN {X 0,Y 222.419,Z 964.272,A -85,B 0,C 180,E1 13612.814,E2 13612.814} C_VEL
LIN {X 0,Y 215.468,Z 969.504,A -85,B 0,C 180,E1 13608.135,E2 13608.135} C_VEL
LIN {X 0,Y 215.244,Z 970.033,A -85,B 0,C 180,E1 13607.569,E2 13607.569} C_VEL
LIN {X 0,Y 214.748,Z 976.652,A -85,B 0,C 180,E1 13598.086,E2 13598.086} C_VEL
LIN {X 0,Y 215.487,Z 977.959,A -85,B 0,C 180,E1 13590.006,E2 13590.006} C_VEL
LIN {X 0,Y 215.135,Z 974.516,A -85,B 0,C 180,E1 13581.941,E2 13581.941} C_VEL
LIN {X 0,Y 215.556,Z 966.243,A -85,B 0,C 180,E1 13573.744,E2 13573.744} C_VEL
LIN {X 0,Y 218.712,Z 950.831,A -85,B 0,C 180,E1 13564.474,E2 13564.474} C_VEL
LIN {X 0,Y 225.579,Z 929.126,A -85,B 0,C 180,E1 13555.77,E2 13555.77} C_VEL
LIN {X 0,Y 235.496,Z 901.488,A -85,B 0,C 180,E1 13548.134,E2 13548.134} C_VEL
LIN {X 0,Y 247.57,Z 867.835,A -85,B 0,C 180,E1 13541.705,E2 13541.705} C_VEL
LIN {X 0,Y 260.716,Z 828.412,A -85,B 0,C 180,E1 13536.604,E2 13536.604} C_VEL
LIN {X 0,Y 264.786,Z 812.991,A -85,B 0,C 180,E1 13535.009,E2 13535.009} C_VEL
LIN {X 0,Y 252.158,Z 776.125,A -85,B 0,C 180,E1 13528.854,E2 13528.854} C_VEL
LIN {X 0,Y 235.974,Z 737.188,A -85,B 0,C 180,E1 13522.074,E2 13522.074} C_VEL
LIN {X 0,Y 227.068,Z 716.643,A -85,B 0,C 180,E1 13518.07,E2 13518.07} C_VEL
LIN {X 0,Y 223.894,Z 701.721,A -85,B 0,C 180,E1 13513.836,E2 13513.836} C_VEL
LIN {X 0,Y 222.176,Z 699.613,A -85,B 0,C 180,E1 13511.765,E2 13511.765} C_VEL
LIN {X 0,Y 218.909,Z 694.321,A -85,B 0,C 180,E1 13505.892,E2 13505.892} C_VEL
LIN {X 0,Y 218.345,Z 692.686,A -85,B 0,C 180,E1 13503.971,E2 13503.971} C_VEL
LIN {X 0,Y 218.691,Z 693.395,A -85,B 0,C 180,E1 13492.818,E2 13492.818} C_VEL
LIN {X 0,Y 221.106,Z 698.941,A -85,B 0,C 180,E1 13487.584,E2 13487.584} C_VEL
LIN {X 0,Y 223.617,Z 701.277,A -85,B 0,C 180,E1 13484.443,E2 13484.443} C_VEL
LIN {X 0,Y 228.801,Z 709.331,A -85,B 0,C 180,E1 13479.321,E2 13479.321} C_VEL
LIN {X 0,Y 237.119,Z 721.404,A -85,B 0,C 180,E1 13473.457,E2 13473.457} C_VEL
LIN {X 0,Y 249.798,Z 742.159,A -85,B 0,C 180,E1 13466.69,E2 13466.69} C_VEL
LIN {X 0,Y 259.407,Z 764.833,A -85,B 0,C 180,E1 13461.306,E2 13461.306} C_VEL
LIN {X 0,Y 264.809,Z 788.196,A -85,B 0,C 180,E1 13456.592,E2 13456.592} C_VEL
LIN {X 0,Y 265.095,Z 796.955,A -85,B 0,C 180,E1 13455.073,E2 13455.073} C_VEL
LIN {X 0,Y 255.949,Z 825.947,A -85,B 0,C 180,E1 13451.264,E2 13451.264} C_VEL
LIN {X 0,Y 245.544,Z 851.393,A -85,B 0,C 180,E1 13446.26,E2 13446.26} C_VEL
LIN {X 0,Y 234.838,Z 873.218,A -85,B 0,C 180,E1 13439.752,E2 13439.752} C_VEL
LIN {X 0,Y 226.339,Z 888.749,A -85,B 0,C 180,E1 13432.536,E2 13432.536} C_VEL
LIN {X 0,Y 220.084,Z 899.959,A -85,B 0,C 180,E1 13423.88,E2 13423.88} C_VEL
LIN {X 0,Y 217.846,Z 904.193,A -85,B 0,C 180,E1 13417.958,E2 13417.958} C_VEL
LIN {X 0,Y 216.994,Z 906.214,A -85,B 0,C 180,E1 13409.994,E2 13409.994} C_VEL
LIN {X 0,Y 217.808,Z 904.266,A -85,B 0,C 180,E1 13402.029,E2 13402.029} C_VEL
LIN {X 0,Y 221.792,Z 896.961,A -85,B 0,C 180,E1 13393.09,E2 13393.09} C_VEL
LIN {X 0,Y 229.109,Z 883.778,A -85,B 0,C 180,E1 13384.644,E2 13384.644} C_VEL
LIN {X 0,Y 238.813,Z 865.534,A -85,B 0,C 180,E1 13377.506,E2 13377.506} C_VEL
LIN {X 0,Y 249.463,Z 842.703,A -85,B 0,C 180,E1 13371.675,E2 13371.675} C_VEL
LIN {X 0,Y 259.896,Z 815.054,A -85,B 0,C 180,E1 13366.999,E2 13366.999} C_VEL
LIN {X 0,Y 265.534,Z 793.978,A -85,B 0,C 180,E1 13364.388,E2 13364.388} C_VEL
LIN {X 0,Y 261.457,Z 771.317,A -85,B 0,C 180,E1 13359.934,E2 13359.934} C_VEL
LIN {X 0,Y 257.989,Z 761.726,A -85,B 0,C 180,E1 13357.745,E2 13357.745} C_VEL
LIN {X 0,Y 247.421,Z 772.157,A -85,B 0,C 180,E1 13355.479,E2 13355.479} C_VEL
LIN {X 0,Y 241.496,Z 781.662,A -85,B 0,C 180,E1 13354.736,E2 13354.736} C_VEL
LIN {X 0,Y 237.277,Z 785.443,A -85,B 0,C 180,E1 13353.525,E2 13353.525} C_VEL
LIN {X 0,Y 232.578,Z 817.847,A -85,B 0,C 180,E1 13350.175,E2 13350.175} C_VEL
LIN {X 0,Y 227.252,Z 846.543,A -85,B 0,C 180,E1 13345.543,E2 13345.543} C_VEL
LIN {X 0,Y 222.407,Z 870.542,A -85,B 0,C 180,E1 13339.82,E2 13339.82} C_VEL
LIN {X 0,Y 218.848,Z 890.345,A -85,B 0,C 180,E1 13332.939,E2 13332.939} C_VEL
LIN {X 0,Y 217.382,Z 905.51,A -85,B 0,C 180,E1 13324.969,E2 13324.969} C_VEL
LIN {X 0,Y 218.255,Z 913.741,A -85,B 0,C 180,E1 13318.01,E2 13318.01} C_VEL
LIN {X 0,Y 220.569,Z 917.642,A -85,B 0,C 180,E1 13312.128,E2 13312.128} C_VEL
LIN {X 0,Y 226.427,Z 918.709,A -85,B 0,C 180,E1 13304.532,E2 13304.532} C_VEL
LIN {X 0,Y 238.834,Z 913.851,A -85,B 0,C 180,E1 13295.746,E2 13295.746} C_VEL
LIN {X 0,Y 256.98,Z 902.824,A -85,B 0,C 180,E1 13288.091,E2 13288.091} C_VEL
LIN {X 0,Y 271.243,Z 893.272,A -85,B 0,C 180,E1 13283.981,E2 13283.981} C_VEL
LIN {X 0,Y 271.308,Z 893.491,A -85,B 0,C 180,E1 13283.451,E2 13283.451} C_VEL
LIN {X 0,Y 244.355,Z 921.545,A -85,B 0,C 180,E1 13275.14,E2 13275.14} C_VEL
LIN {X 0,Y 225.323,Z 947.345,A -85,B 0,C 180,E1 13263.886,E2 13263.886} C_VEL
LIN {X 0,Y 216.748,Z 964.693,A -85,B 0,C 180,E1 13252.522,E2 13252.522} C_VEL
LIN {X 0,Y 215.244,Z 970.033,A -85,B 0,C 180,E1 13247.569,E2 13247.569} C_VEL
LIN {X 0,Y 212.373,Z 972.716,A -85,B 0,C 180,E1 13244.21,E2 13244.21} C_VEL
LIN {X 0,Y 206.923,Z 975.268,A -85,B 0,C 180,E1 13238.39,E2 13238.39} C_VEL
LIN {X 0,Y 207.726,Z 976.445,A -85,B 0,C 180,E1 13230.006,E2 13230.006} C_VEL
LIN {X 0,Y 207.369,Z 972.752,A -85,B 0,C 180,E1 13221.638,E2 13221.638} C_VEL
LIN {X 0,Y 207.9,Z 964.145,A -85,B 0,C 180,E1 13213.128,E2 13213.128} C_VEL
LIN {X 0,Y 211.304,Z 948.873,A -85,B 0,C 180,E1 13203.511,E2 13203.511} C_VEL
LIN {X 0,Y 218.038,Z 928.857,A -85,B 0,C 180,E1 13195.188,E2 13195.188} C_VEL
LIN {X 0,Y 227.269,Z 903.192,A -85,B 0,C 180,E1 13188.029,E2 13188.029} C_VEL
LIN {X 0,Y 240.136,Z 868.078,A -85,B 0,C 180,E1 13181.06,E2 13181.06} C_VEL
LIN {X 0,Y 253.523,Z 829.162,A -85,B 0,C 180,E1 13175.851,E2 13175.851} C_VEL
LIN {X 0,Y 257.499,Z 815.039,A -85,B 0,C 180,E1 13174.352,E2 13174.352} C_VEL
LIN {X 0,Y 245.154,Z 778.418,A -85,B 0,C 180,E1 13167.998,E2 13167.998} C_VEL
LIN {X 0,Y 229.544,Z 740.28,A -85,B 0,C 180,E1 13161.078,E2 13161.078} C_VEL
LIN {X 0,Y 224.898,Z 723.353,A -85,B 0,C 180,E1 13157.089,E2 13157.089} C_VEL
LIN {X 0,Y 221.935,Z 707.918,A -85,B 0,C 180,E1 13152.648,E2 13152.648} C_VEL
LIN {X 0,Y 217.893,Z 702.643,A -85,B 0,C 180,E1 13145.92,E2 13145.92} C_VEL
LIN {X 0,Y 217.385,Z 700.531,A -85,B 0,C 180,E1 13143.989,E2 13143.989} C_VEL
LIN {X 0,Y 217.55,Z 701.392,A -85,B 0,C 180,E1 13133.205,E2 13133.205} C_VEL
LIN {X 0,Y 220.73,Z 707.331,A -85,B 0,C 180,E1 13126.744,E2 13126.744} C_VEL
LIN {X 0,Y 222.369,Z 709.614,A -85,B 0,C 180,E1 13124.633,E2 13124.633} C_VEL
LIN {X 0,Y 227.044,Z 716.829,A -85,B 0,C 180,E1 13119.879,E2 13119.879} C_VEL
LIN {X 0,Y 235.207,Z 729.201,A -85,B 0,C 180,E1 13113.894,E2 13113.894} C_VEL
LIN {X 0,Y 246.182,Z 748.093,A -85,B 0,C 180,E1 13107.577,E2 13107.577} C_VEL
LIN {X 0,Y 254.517,Z 769.142,A -85,B 0,C 180,E1 13102.336,E2 13102.336} C_VEL
LIN {X 0,Y 259.178,Z 791.409,A -85,B 0,C 180,E1 13097.617,E2 13097.617} C_VEL
LIN {X 0,Y 259.112,Z 800.232,A -85,B 0,C 180,E1 13096.071,E2 13096.071} C_VEL
LIN {X 0,Y 249.219,Z 829.598,A -85,B 0,C 180,E1 13092.049,E2 13092.049} C_VEL
LIN {X 0,Y 238.476,Z 854.302,A -85,B 0,C 180,E1 13086.946,E2 13086.946} C_VEL
LIN {X 0,Y 228.053,Z 874.559,A -85,B 0,C 180,E1 13080.686,E2 13080.686} C_VEL
LIN {X 0,Y 219.127,Z 890.001,A -85,B 0,C 180,E1 13073.321,E2 13073.321} C_VEL
LIN {X 0,Y 212.51,Z 901.208,A -85,B 0,C 180,E1 13064.385,E2 13064.385} C_VEL
LIN {X 0,Y 210.125,Z 905.44,A -85,B 0,C 180,E1 13058.252,E2 13058.252} C_VEL
LIN {X 0,Y 209.203,Z 907.459,A -85,B 0,C 180,E1 13049.994,E2 13049.994} C_VEL
LIN {X 0,Y 210.095,Z 905.511,A -85,B 0,C 180,E1 13041.734,E2 13041.734} C_VEL
LIN {X 0,Y 214.315,Z 898.211,A -85,B 0,C 180,E1 13032.482,E2 13032.482} C_VEL
LIN {X 0,Y 222.091,Z 885.021,A -85,B 0,C 180,E1 13023.783,E2 13023.783} C_VEL
LIN {X 0,Y 232.275,Z 866.775,A -85,B 0,C 180,E1 13016.472,E2 13016.472} C_VEL
LIN {X 0,Y 243.217,Z 844.363,A -85,B 0,C 180,E1 13010.625,E2 13010.625} C_VEL
LIN {X 0,Y 253.797,Z 817.496,A -85,B 0,C 180,E1 13005.97,E2 13005.97} C_VEL
LIN {X 0,Y 259.75,Z 796.351,A -85,B 0,C 180,E1 13003.259,E2 13003.259} C_VEL
LIN {X 0,Y 256.091,Z 774.451,A -85,B 0,C 180,E1 12998.721,E2 12998.721} C_VEL
LIN {X 0,Y 255.517,Z 772.462,A -85,B 0,C 180,E1 12998.275,E2 12998.275} C_VEL
LIN {X 0,Y 251.791,Z 774.465,A -85,B 0,C 180,E1 12997.336,E2 12997.336} C_VEL
LIN {X 0,Y 248.28,Z 779.156,A -85,B 0,C 180,E1 12996.816,E2 12996.816} C_VEL
LIN {X 0,Y 241.494,Z 788.101,A -85,B 0,C 180,E1 12995.887,E2 12995.887} C_VEL
LIN {X 0,Y 236.899,Z 792.462,A -85,B 0,C 180,E1 12994.966,E2 12994.966} C_VEL
LIN {X 0,Y 230.391,Z 799.661,A -85,B 0,C 180,E1 12993.816,E2 12993.816} C_VEL
LIN {X 0,Y 228.004,Z 801.131,A -85,B 0,C 180,E1 12992.939,E2 12992.939} C_VEL
LIN {X 0,Y 222.767,Z 832.199,A -85,B 0,C 180,E1 12988.845,E2 12988.845} C_VEL
LIN {X 0,Y 217.049,Z 859.866,A -85,B 0,C 180,E1 12983.28,E2 12983.28} C_VEL
LIN {X 0,Y 212.468,Z 882.664,A -85,B 0,C 180,E1 12976.494,E2 12976.494} C_VEL
LIN {X 0,Y 209.971,Z 899.187,A -85,B 0,C 180,E1 12969.296,E2 12969.296} C_VEL
LIN {X 0,Y 209.863,Z 911.588,A -85,B 0,C 180,E1 12961.021,E2 12961.021} C_VEL
LIN {X 0,Y 212.879,Z 919.055,A -85,B 0,C 180,E1 12951.841,E2 12951.841} C_VEL
LIN {X 0,Y 219.054,Z 920.637,A -85,B 0,C 180,E1 12943.998,E2 12943.998} C_VEL
LIN {X 0,Y 232.119,Z 916.66,A -85,B 0,C 180,E1 12934.997,E2 12934.997} C_VEL
LIN {X 0,Y 251.052,Z 906.721,A -85,B 0,C 180,E1 12927.245,E2 12927.245} C_VEL
LIN {X 0,Y 260.207,Z 901.357,A -85,B 0,C 180,E1 12924.549,E2 12924.549} C_VEL
LIN {X 0,Y 262.209,Z 900.319,A -85,B 0,C 180,E1 12923.69,E2 12923.69} C_VEL
LIN {X 0,Y 233.164,Z 928.572,A -85,B 0,C 180,E1 12914.096,E2 12914.096} C_VEL
LIN {X 0,Y 214.656,Z 952.96,A -85,B 0,C 180,E1 12901.474,E2 12901.474} C_VEL
LIN {X 0,Y 207.78,Z 968.026,A -85,B 0,C 180,E1 12889.23,E2 12889.23} C_VEL
LIN {X 0,Y 206.817,Z 974.291,A -85,B 0,C 180,E1 12880.563,E2 12880.563} C_VEL
LIN {X 0,Y 206.923,Z 975.268,A -85,B 0,C 180,E1 12878.39,E2 12878.39} C_VEL
LIN {X 0,Y 204.675,Z 975.849,A -85,B 0,C 180,E1 12874.8,E2 12874.8} C_VEL
LIN {X 0,Y 199.787,Z 974.422,A -85,B 0,C 180,E1 12868.684,E2 12868.684} C_VEL
LIN {X 0,Y 199.628,Z 970.886,A -85,B 0,C 180,E1 12861.311,E2 12861.311} C_VEL
LIN {X 0,Y 200.458,Z 960.787,A -85,B 0,C 180,E1 12850.949,E2 12850.949} C_VEL
LIN {X 0,Y 204.193,Z 946.64,A -85,B 0,C 180,E1 12842.01,E2 12842.01} C_VEL
LIN {X 0,Y 211.829,Z 925.985,A -85,B 0,C 180,E1 12833.378,E2 12833.378} C_VEL
LIN {X 0,Y 221.518,Z 900.894,A -85,B 0,C 180,E1 12826.353,E2 12826.353} C_VEL
LIN {X 0,Y 231.632,Z 871.748,A -85,B 0,C 180,E1 12820.878,E2 12820.878} C_VEL
LIN {X 0,Y 246.878,Z 828.111,A -85,B 0,C 180,E1 12814.881,E2 12814.881} C_VEL
LIN {X 0,Y 249.882,Z 815.785,A -85,B 0,C 180,E1 12813.459,E2 12813.459} C_VEL
LIN {X 0,Y 237.672,Z 779.548,A -85,B 0,C 180,E1 12806.903,E2 12806.903} C_VEL
LIN {X 0,Y 227.714,Z 752.706,A -85,B 0,C 180,E1 12801.623,E2 12801.623} C_VEL
LIN {X 0,Y 220.482,Z 715.662,A -85,B 0,C 180,E1 12792.13,E2 12792.13} C_VEL
LIN {X 0,Y 216.646,Z 709.818,A -85,B 0,C 180,E1 12785.088,E2 12785.088} C_VEL
LIN {X 0,Y 216.425,Z 708.374,A -85,B 0,C 180,E1 12784.007,E2 12784.007} C_VEL
LIN {X 0,Y 216.42,Z 709.085,A -85,B 0,C 180,E1 12773.703,E2 12773.703} C_VEL
LIN {X 0,Y 219.788,Z 715.211,A -85,B 0,C 180,E1 12766.686,E2 12766.686} C_VEL
LIN {X 0,Y 225.314,Z 724.291,A -85,B 0,C 180,E1 12760.446,E2 12760.446} C_VEL
LIN {X 0,Y 233.6,Z 737.409,A -85,B 0,C 180,E1 12754.153,E2 12754.153} C_VEL
LIN {X 0,Y 243.367,Z 755.884,A -85,B 0,C 180,E1 12747.945,E2 12747.945} C_VEL
LIN {X 0,Y 250.403,Z 776.444,A -85,B 0,C 180,E1 12742.684,E2 12742.684} C_VEL
LIN {X 0,Y 253.939,Z 798.862,A -85,B 0,C 180,E1 12737.776,E2 12737.776} C_VEL
LIN {X 0,Y 246.146,Z 824.185,A -85,B 0,C 180,E1 12734.348,E2 12734.348} C_VEL
LIN {X 0,Y 234.673,Z 850.684,A -85,B 0,C 180,E1 12729.302,E2 12729.302} C_VEL
LIN {X 0,Y 222.982,Z 872.959,A -85,B 0,C 180,E1 12722.773,E2 12722.773} C_VEL
LIN {X 0,Y 212.991,Z 889.632,A -85,B 0,C 180,E1 12715.151,E2 12715.151} C_VEL
LIN {X 0,Y 206.157,Z 900.498,A -85,B 0,C 180,E1 12707.019,E2 12707.019} C_VEL
LIN {X 0,Y 202.405,Z 906.689,A -85,B 0,C 180,E1 12698.569,E2 12698.569} C_VEL
LIN {X 0,Y 201.419,Z 908.704,A -85,B 0,C 180,E1 12689.993,E2 12689.993} C_VEL
LIN {X 0,Y 202.377,Z 906.758,A -85,B 0,C 180,E1 12681.417,E2 12681.417} C_VEL
LIN {X 0,Y 206.947,Z 899.376,A -85,B 0,C 180,E1 12671.754,E2 12671.754} C_VEL
LIN {X 0,Y 215.124,Z 886.264,A -85,B 0,C 180,E1 12662.866,E2 12662.866} C_VEL
LIN {X 0,Y 225.8,Z 868.017,A -85,B 0,C 180,E1 12655.377,E2 12655.377} C_VEL
LIN {X 0,Y 237.424,Z 845.166,A -85,B 0,C 180,E1 12649.338,E2 12649.338} C_VEL
LIN {X 0,Y 248.485,Z 818.163,A -85,B 0,C 180,E1 12644.645,E2 12644.645} C_VEL
LIN {X 0,Y 254.085,Z 799.317,A -85,B 0,C 180,E1 12642.194,E2 12642.194} C_VEL
LIN {X 0,Y 251.763,Z 781.764,A -85,B 0,C 180,E1 12638.417,E2 12638.417} C_VEL
LIN {X 0,Y 242.78,Z 793.02,A -85,B 0,C 180,E1 12637.316,E2 12637.316} C_VEL
LIN {X 0,Y 229.753,Z 805.733,A -85,B 0,C 180,E1 12635.064,E2 12635.064} C_VEL
LIN {X 0,Y 220.802,Z 813.291,A -85,B 0,C 180,E1 12633.13,E2 12633.13} C_VEL
LIN {X 0,Y 218.788,Z 814,A -85,B 0,C 180,E1 12632.298,E2 12632.298} C_VEL
LIN {X 0,Y 212.951,Z 844.121,A -85,B 0,C 180,E1 12627.461,E2 12627.461} C_VEL
LIN {X 0,Y 207.46,Z 869.685,A -85,B 0,C 180,E1 12621.315,E2 12621.315} C_VEL
LIN {X 0,Y 203.363,Z 891.017,A -85,B 0,C 180,E1 12613.751,E2 12613.751} C_VEL
LIN {X 0,Y 201.707,Z 906.709,A -85,B 0,C 180,E1 12605.356,E2 12605.356} C_VEL
LIN {X 0,Y 202.601,Z 915.766,A -85,B 0,C 180,E1 12597.856,E2 12597.856} C_VEL
LIN {X 0,Y 205.202,Z 920.428,A -85,B 0,C 180,E1 12591.534,E2 12591.534} C_VEL
LIN {X 0,Y 211.718,Z 922.555,A -85,B 0,C 180,E1 12583.427,E2 12583.427} C_VEL
LIN {X 0,Y 225.409,Z 919.382,A -85,B 0,C 180,E1 12574.199,E2 12574.199} C_VEL
LIN {X 0,Y 247.496,Z 909.346,A -85,B 0,C 180,E1 12565.634,E2 12565.634} C_VEL
LIN {X 0,Y 252.188,Z 906.951,A -85,B 0,C 180,E1 12564.305,E2 12564.305} C_VEL
LIN {X 0,Y 252.321,Z 907.197,A -85,B 0,C 180,E1 12563.725,E2 12563.725} C_VEL
LIN {X 0,Y 221.975,Z 934.936,A -85,B 0,C 180,E1 12552.839,E2 12552.839} C_VEL
LIN {X 0,Y 205.182,Z 956.276,A -85,B 0,C 180,E1 12539.828,E2 12539.828} C_VEL
LIN {X 0,Y 199.513,Z 968.851,A -85,B 0,C 180,E1 12527.618,E2 12527.618} C_VEL
LIN {X 0,Y 199.084,Z 973.947,A -85,B 0,C 180,E1 12518.393,E2 12518.393} C_VEL
LIN {X 0,Y 200.001,Z 974.845,A -85,B 0,C 180,E1 12510.007,E2 12510.007} C_VEL
LIN {X 0,Y 199.787,Z 974.422,A -85,B 0,C 180,E1 12508.684,E2 12508.684} C_VEL
LIN {X 0,Y 197.133,Z 972.597,A -85,B 0,C 180,E1 12505.014,E2 12505.014} C_VEL
LIN {X 0,Y 191.807,Z 967.672,A -85,B 0,C 180,E1 12498.814,E2 12498.814} C_VEL
LIN {X 0,Y 192.807,Z 959.2,A -85,B 0,C 180,E1 12489.93,E2 12489.93} C_VEL
LIN {X 0,Y 197.418,Z 944.06,A -85,B 0,C 180,E1 12480.215,E2 12480.215} C_VEL
LIN {X 0,Y 205.799,Z 923.092,A -85,B 0,C 180,E1 12471.452,E2 12471.452} C_VEL
LIN {X 0,Y 216.242,Z 897.74,A -85,B 0,C 180,E1 12464.408,E2 12464.408} C_VEL
LIN {X 0,Y 227.253,Z 867.692,A -85,B 0,C 180,E1 12458.88,E2 12458.88} C_VEL
LIN {X 0,Y 242.826,Z 818.516,A -85,B 0,C 180,E1 12452.909,E2 12452.909} C_VEL
LIN {X 0,Y 229.856,Z 777.357,A -85,B 0,C 180,E1 12444.763,E2 12444.763} C_VEL
LIN {X 0,Y 218.903,Z 723.422,A -85,B 0,C 180,E1 12431.439,E2 12431.439} C_VEL
LIN {X 0,Y 215.39,Z 716.5,A -85,B 0,C 180,E1 12423.9,E2 12423.9} C_VEL
LIN {X 0,Y 215.302,Z 716.67,A -85,B 0,C 180,E1 12414.259,E2 12414.259} C_VEL
LIN {X 0,Y 218.543,Z 722.922,A -85,B 0,C 180,E1 12407.023,E2 12407.023} C_VEL
LIN {X 0,Y 223.814,Z 732.115,A -85,B 0,C 180,E1 12400.822,E2 12400.822} C_VEL
LIN {X 0,Y 232.429,Z 746.28,A -85,B 0,C 180,E1 12394.021,E2 12394.021} C_VEL
LIN {X 0,Y 241.309,Z 766.311,A -85,B 0,C 180,E1 12387.506,E2 12387.506} C_VEL
LIN {X 0,Y 246.687,Z 786.794,A -85,B 0,C 180,E1 12382.301,E2 12382.301} C_VEL
LIN {X 0,Y 248.145,Z 804.014,A -85,B 0,C 180,E1 12378.501,E2 12378.501} C_VEL
LIN {X 0,Y 237.407,Z 833.276,A -85,B 0,C 180,E1 12374.356,E2 12374.356} C_VEL
LIN {X 0,Y 225.679,Z 857.78,A -85,B 0,C 180,E1 12369.063,E2 12369.063} C_VEL
LIN {X 0,Y 213.536,Z 878.946,A -85,B 0,C 180,E1 12362.029,E2 12362.029} C_VEL
LIN {X 0,Y 203.844,Z 894.109,A -85,B 0,C 180,E1 12354.02,E2 12354.02} C_VEL
LIN {X 0,Y 197.402,Z 903.709,A -85,B 0,C 180,E1 12345.512,E2 12345.512} C_VEL
LIN {X 0,Y 194.697,Z 907.936,A -85,B 0,C 180,E1 12338.911,E2 12338.911} C_VEL
LIN {X 0,Y 193.622,Z 909.951,A -85,B 0,C 180,E1 12329.993,E2 12329.993} C_VEL
LIN {X 0,Y 195.453,Z 906.891,A -85,B 0,C 180,E1 12318.864,E2 12318.864} C_VEL
LIN {X 0,Y 201.014,Z 898.391,A -85,B 0,C 180,E1 12309.093,E2 12309.093} C_VEL
LIN {X 0,Y 210.039,Z 884.607,A -85,B 0,C 180,E1 12300.392,E2 12300.392} C_VEL
LIN {X 0,Y 221.876,Z 865.012,A -85,B 0,C 180,E1 12292.862,E2 12292.862} C_VEL
LIN {X 0,Y 233.99,Z 841.386,A -85,B 0,C 180,E1 12287.054,E2 12287.054} C_VEL
LIN {X 0,Y 244.906,Z 814.096,A -85,B 0,C 180,E1 12282.608,E2 12282.608} C_VEL
LIN {X 0,Y 248.455,Z 801.707,A -85,B 0,C 180,E1 12280.951,E2 12280.951} C_VEL
LIN {X 0,Y 247.516,Z 794.406,A -85,B 0,C 180,E1 12279.201,E2 12279.201} C_VEL
LIN {X 0,Y 230.72,Z 810.444,A -85,B 0,C 180,E1 12276.698,E2 12276.698} C_VEL
LIN {X 0,Y 219.609,Z 819.255,A -85,B 0,C 180,E1 12274.441,E2 12274.441} C_VEL
LIN {X 0,Y 210.225,Z 825.669,A -85,B 0,C 180,E1 12271.95,E2 12271.95} C_VEL
LIN {X 0,Y 209.374,Z 825.816,A -85,B 0,C 180,E1 12271.488,E2 12271.488} C_VEL
LIN {X 0,Y 203.453,Z 853.917,A -85,B 0,C 180,E1 12266.115,E2 12266.115} C_VEL
LIN {X 0,Y 197.864,Z 879.241,A -85,B 0,C 180,E1 12258.901,E2 12258.901} C_VEL
LIN {X 0,Y 194.489,Z 898.666,A -85,B 0,C 180,E1 12250.608,E2 12250.608} C_VEL
LIN {X 0,Y 193.943,Z 911.798,A -85,B 0,C 180,E1 12242.219,E2 12242.219} C_VEL
LIN {X 0,Y 196.292,Z 920.335,A -85,B 0,C 180,E1 12233.369,E2 12233.369} C_VEL
LIN {X 0,Y 200.37,Z 923.615,A -85,B 0,C 180,E1 12226.934,E2 12226.934} C_VEL
LIN {X 0,Y 209.333,Z 924.232,A -85,B 0,C 180,E1 12218.865,E2 12218.865} C_VEL
LIN {X 0,Y 226.268,Z 919.563,A -85,B 0,C 180,E1 12209.981,E2 12209.981} C_VEL
LIN {X 0,Y 239.301,Z 914.285,A -85,B 0,C 180,E1 12205.416,E2 12205.416} C_VEL
LIN {X 0,Y 242.812,Z 913.019,A -85,B 0,C 180,E1 12203.905,E2 12203.905} C_VEL
LIN {X 0,Y 211.183,Z 940.117,A -85,B 0,C 180,E1 12191.649,E2 12191.649} C_VEL
LIN {X 0,Y 195.554,Z 959.452,A -85,B 0,C 180,E1 12177.59,E2 12177.59} C_VEL
LIN {X 0,Y 191.374,Z 969.164,A -85,B 0,C 180,E1 12166.028,E2 12166.028} C_VEL
LIN {X 0,Y 191.284,Z 972.46,A -85,B 0,C 180,E1 12159.085,E2 12159.085} C_VEL
LIN {X 0,Y 192.276,Z 973.217,A -85,B 0,C 180,E1 12150.007,E2 12150.007} C_VEL
LIN {X 0,Y 191.861,Z 969.025,A -85,B 0,C 180,E1 12140.956,E2 12140.956} C_VEL
LIN {X 0,Y 191.807,Z 967.672,A -85,B 0,C 180,E1 12138.814,E2 12138.814} C_VEL
LIN {X 0,Y 189.372,Z 964.415,A -85,B 0,C 180,E1 12135.056,E2 12135.056} C_VEL
LIN {X 0,Y 185.11,Z 958.297,A -85,B 0,C 180,E1 12129.398,E2 12129.398} C_VEL
LIN {X 0,Y 185.199,Z 957.516,A -85,B 0,C 180,E1 12128.759,E2 12128.759} C_VEL
LIN {X 0,Y 190.696,Z 941.665,A -85,B 0,C 180,E1 12118.389,E2 12118.389} C_VEL
LIN {X 0,Y 199.853,Z 920.487,A -85,B 0,C 180,E1 12109.506,E2 12109.506} C_VEL
LIN {X 0,Y 210.995,Z 895.206,A -85,B 0,C 180,E1 12102.518,E2 12102.518} C_VEL
LIN {X 0,Y 222.562,Z 865.141,A -85,B 0,C 180,E1 12097.04,E2 12097.04} C_VEL
LIN {X 0,Y 232.422,Z 832.664,A -85,B 0,C 180,E1 12093.282,E2 12093.282} C_VEL
LIN {X 0,Y 235.39,Z 820.088,A -85,B 0,C 180,E1 12092.154,E2 12092.154} C_VEL
LIN {X 0,Y 225.539,Z 778.202,A -85,B 0,C 180,E1 12082.503,E2 12082.503} C_VEL
LIN {X 0,Y 217.265,Z 730.508,A -85,B 0,C 180,E1 12070.513,E2 12070.513} C_VEL
LIN {X 0,Y 214.313,Z 724.337,A -85,B 0,C 180,E1 12063.541,E2 12063.541} C_VEL
LIN {X 0,Y 214.231,Z 724.527,A -85,B 0,C 180,E1 12054.607,E2 12054.607} C_VEL
LIN {X 0,Y 218.163,Z 732.635,A -85,B 0,C 180,E1 12046.022,E2 12046.022} C_VEL
LIN {X 0,Y 224.39,Z 742.919,A -85,B 0,C 180,E1 12039.337,E2 12039.337} C_VEL
LIN {X 0,Y 232.673,Z 759.737,A -85,B 0,C 180,E1 12032.359,E2 12032.359} C_VEL
LIN {X 0,Y 239.194,Z 778.651,A -85,B 0,C 180,E1 12026.497,E2 12026.497} C_VEL
LIN {X 0,Y 242.571,Z 799.555,A -85,B 0,C 180,E1 12021.26,E2 12021.26} C_VEL
LIN {X 0,Y 242.336,Z 807.363,A -85,B 0,C 180,E1 12019.629,E2 12019.629} C_VEL
LIN {X 0,Y 231.376,Z 835.648,A -85,B 0,C 180,E1 12015.501,E2 12015.501} C_VEL
LIN {X 0,Y 218.958,Z 860.349,A -85,B 0,C 180,E1 12009.991,E2 12009.991} C_VEL
LIN {X 0,Y 206.951,Z 880.195,A -85,B 0,C 180,E1 12003.177,E2 12003.177} C_VEL
LIN {X 0,Y 196.725,Z 895.359,A -85,B 0,C 180,E1 11994.948,E2 11994.948} C_VEL
LIN {X 0,Y 189.887,Z 904.959,A -85,B 0,C 180,E1 11986.143,E2 11986.143} C_VEL
LIN {X 0,Y 186.991,Z 909.185,A -85,B 0,C 180,E1 11979.281,E2 11979.281} C_VEL
LIN {X 0,Y 185.837,Z 911.196,A -85,B 0,C 180,E1 11969.993,E2 11969.993} C_VEL
LIN {X 0,Y 187.793,Z 908.14,A -85,B 0,C 180,E1 11958.403,E2 11958.403} C_VEL
LIN {X 0,Y 193.746,Z 899.618,A -85,B 0,C 180,E1 11948.25,E2 11948.25} C_VEL
LIN {X 0,Y 203.292,Z 885.85,A -85,B 0,C 180,E1 11939.306,E2 11939.306} C_VEL
LIN {X 0,Y 215.698,Z 866.254,A -85,B 0,C 180,E1 11931.609,E2 11931.609} C_VEL
LIN {X 0,Y 228.34,Z 842.621,A -85,B 0,C 180,E1 11925.72,E2 11925.72} C_VEL
LIN {X 0,Y 239.793,Z 815.098,A -85,B 0,C 180,E1 11921.211,E2 11921.211} C_VEL
LIN {X 0,Y 242.936,Z 805.116,A -85,B 0,C 180,E1 11919.884,E2 11919.884} C_VEL
LIN {X 0,Y 228.243,Z 817.52,A -85,B 0,C 180,E1 11917.655,E2 11917.655} C_VEL
LIN {X 0,Y 217.289,Z 825.657,A -85,B 0,C 180,E1 11915.509,E2 11915.509} C_VEL
LIN {X 0,Y 201.927,Z 835.81,A -85,B 0,C 180,E1 11911.527,E2 11911.527} C_VEL
LIN {X 0,Y 199.885,Z 836.643,A -85,B 0,C 180,E1 11910.497,E2 11910.497} C_VEL
LIN {X 0,Y 193.568,Z 864.522,A -85,B 0,C 180,E1 11904.146,E2 11904.146} C_VEL
LIN {X 0,Y 188.663,Z 887.021,A -85,B 0,C 180,E1 11896.514,E2 11896.514} C_VEL
LIN {X 0,Y 186.217,Z 903.928,A -85,B 0,C 180,E1 11888.141,E2 11888.141} C_VEL
LIN {X 0,Y 186.684,Z 916.345,A -85,B 0,C 180,E1 11878.832,E2 11878.832} C_VEL
LIN {X 0,Y 191.208,Z 924.177,A -85,B 0,C 180,E1 11868.612,E2 11868.612} C_VEL
LIN {X 0,Y 202.272,Z 926.32,A -85,B 0,C 180,E1 11858.09,E2 11858.09} C_VEL
LIN {X 0,Y 219.968,Z 922.604,A -85,B 0,C 180,E1 11849.028,E2 11849.028} C_VEL
LIN {X 0,Y 233.493,Z 917.989,A -85,B 0,C 180,E1 11844.427,E2 11844.427} C_VEL
LIN {X 0,Y 198.422,Z 946.665,A -85,B 0,C 180,E1 11828.87,E2 11828.87} C_VEL
LIN {X 0,Y 185.613,Z 962.853,A -85,B 0,C 180,E1 11813.994,E2 11813.994} C_VEL
LIN {X 0,Y 183.425,Z 969.136,A -85,B 0,C 180,E1 11804.297,E2 11804.297} C_VEL
LIN {X 0,Y 183.837,Z 971.782,A -85,B 0,C 180,E1 11794.716,E2 11794.716} C_VEL
LIN {X 0,Y 184.544,Z 971.555,A -85,B 0,C 180,E1 11790.007,E2 11790.007} C_VEL
LIN {X 0,Y 183.968,Z 967.322,A -85,B 0,C 180,E1 11779.867,E2 11779.867} C_VEL
LIN {X 0,Y 184.917,Z 958.942,A -85,B 0,C 180,E1 11769.997,E2 11769.997} C_VEL
LIN {X 0,Y 185.199,Z 957.516,A -85,B 0,C 180,E1 11768.759,E2 11768.759} C_VEL
LIN {X 0,Y 183.311,Z 950.961,A -85,B 0,C 180,E1 11763.738,E2 11763.738} C_VEL
LIN {X 0,Y 182.344,Z 943.392,A -85,B 0,C 180,E1 11758.764,E2 11758.764} C_VEL
LIN {X 0,Y 191.712,Z 923.167,A -85,B 0,C 180,E1 11749.338,E2 11749.338} C_VEL
LIN {X 0,Y 203.363,Z 898.558,A -85,B 0,C 180,E1 11741.907,E2 11741.907} C_VEL
LIN {X 0,Y 215.685,Z 869.217,A -85,B 0,C 180,E1 11736.132,E2 11736.132} C_VEL
LIN {X 0,Y 226.288,Z 837.845,A -85,B 0,C 180,E1 11732.198,E2 11732.198} C_VEL
LIN {X 0,Y 229.88,Z 824.232,A -85,B 0,C 180,E1 11730.974,E2 11730.974} C_VEL
LIN {X 0,Y 223.006,Z 787.065,A -85,B 0,C 180,E1 11722.118,E2 11722.118} C_VEL
LIN {X 0,Y 215.653,Z 737.868,A -85,B 0,C 180,E1 11709.574,E2 11709.574} C_VEL
LIN {X 0,Y 213.029,Z 731.737,A -85,B 0,C 180,E1 11702.039,E2 11702.039} C_VEL
LIN {X 0,Y 213.192,Z 732.539,A -85,B 0,C 180,E1 11694.796,E2 11694.796} C_VEL
LIN {X 0,Y 216.855,Z 740.352,A -85,B 0,C 180,E1 11686.414,E2 11686.414} C_VEL
LIN {X 0,Y 222.53,Z 750.631,A -85,B 0,C 180,E1 11679.804,E2 11679.804} C_VEL
LIN {X 0,Y 229.562,Z 766.571,A -85,B 0,C 180,E1 11673.013,E2 11673.013} C_VEL
LIN {X 0,Y 234.867,Z 784.346,A -85,B 0,C 180,E1 11667.309,E2 11667.309} C_VEL
LIN {X 0,Y 237.364,Z 805.096,A -85,B 0,C 180,E1 11661.915,E2 11661.915} C_VEL
LIN {X 0,Y 236.676,Z 810.641,A -85,B 0,C 180,E1 11660.812,E2 11660.812} C_VEL
LIN {X 0,Y 224.928,Z 839.082,A -85,B 0,C 180,E1 11656.496,E2 11656.496} C_VEL
LIN {X 0,Y 211.935,Z 863.509,A -85,B 0,C 180,E1 11650.792,E2 11650.792} C_VEL
LIN {X 0,Y 199.341,Z 883.118,A -85,B 0,C 180,E1 11643.648,E2 11643.648} C_VEL
LIN {X 0,Y 188.572,Z 898.037,A -85,B 0,C 180,E1 11634.836,E2 11634.836} C_VEL
LIN {X 0,Y 181.217,Z 907.889,A -85,B 0,C 180,E1 11624.46,E2 11624.46} C_VEL
LIN {X 0,Y 178.289,Z 911.909,A -85,B 0,C 180,E1 11614.848,E2 11614.848} C_VEL
LIN {X 0,Y 178.284,Z 911.936,A -85,B 0,C 180,E1 11605.137,E2 11605.137} C_VEL
LIN {X 0,Y 181.211,Z 907.966,A -85,B 0,C 180,E1 11595.525,E2 11595.525} C_VEL
LIN {X 0,Y 188.549,Z 898.189,A -85,B 0,C 180,E1 11585.146,E2 11585.146} C_VEL
LIN {X 0,Y 199.143,Z 883.6,A -85,B 0,C 180,E1 11576.437,E2 11576.437} C_VEL
LIN {X 0,Y 212.402,Z 862.929,A -85,B 0,C 180,E1 11568.9,E2 11568.9} C_VEL
LIN {X 0,Y 225.929,Z 837.339,A -85,B 0,C 180,E1 11563.058,E2 11563.058} C_VEL
LIN {X 0,Y 233.372,Z 819.949,A -85,B 0,C 180,E1 11560.271,E2 11560.271} C_VEL
LIN {X 0,Y 227.724,Z 823.041,A -85,B 0,C 180,E1 11559.069,E2 11559.069} C_VEL
LIN {X 0,Y 211.42,Z 834.469,A -85,B 0,C 180,E1 11556.06,E2 11556.06} C_VEL
LIN {X 0,Y 191.061,Z 846.037,A -85,B 0,C 180,E1 11549.922,E2 11549.922} C_VEL
LIN {X 0,Y 189.981,Z 847.868,A -85,B 0,C 180,E1 11549.086,E2 11549.086} C_VEL
LIN {X 0,Y 184.001,Z 873.027,A -85,B 0,C 180,E1 11542.277,E2 11542.277} C_VEL
LIN {X 0,Y 179.644,Z 893.983,A -85,B 0,C 180,E1 11533.963,E2 11533.963} C_VEL
LIN {X 0,Y 178.153,Z 909.656,A -85,B 0,C 180,E1 11524.848,E2 11524.848} C_VEL
LIN {X 0,Y 179.776,Z 920.516,A -85,B 0,C 180,E1 11515.175,E2 11515.175} C_VEL
LIN {X 0,Y 185.324,Z 926.575,A -85,B 0,C 180,E1 11505.852,E2 11505.852} C_VEL
LIN {X 0,Y 195.246,Z 928.409,A -85,B 0,C 180,E1 11497.258,E2 11497.258} C_VEL
LIN {X 0,Y 212.023,Z 925.973,A -85,B 0,C 180,E1 11488.673,E2 11488.673} C_VEL
LIN {X 0,Y 223.378,Z 923.191,A -85,B 0,C 180,E1 11484.173,E2 11484.173} C_VEL
LIN {X 0,Y 192.016,Z 946.435,A -85,B 0,C 180,E1 11470.351,E2 11470.351} C_VEL
LIN {X 0,Y 178.138,Z 961.763,A -85,B 0,C 180,E1 11455.068,E2 11455.068} C_VEL
LIN {X 0,Y 175.621,Z 967.721,A -85,B 0,C 180,E1 11444.946,E2 11444.946} C_VEL
LIN {X 0,Y 176.042,Z 970.133,A -85,B 0,C 180,E1 11434.925,E2 11434.925} C_VEL
LIN {X 0,Y 176.82,Z 969.782,A -85,B 0,C 180,E1 11430.007,E2 11430.007} C_VEL
LIN {X 0,Y 176.145,Z 966.465,A -85,B 0,C 180,E1 11420.142,E2 11420.142} C_VEL
LIN {X 0,Y 177.089,Z 958.185,A -85,B 0,C 180,E1 11409.625,E2 11409.625} C_VEL
LIN {X 0,Y 182.344,Z 943.392,A -85,B 0,C 180,E1 11398.764,E2 11398.764} C_VEL
LIN {X 0,Y 182.357,Z 935.057,A -85,B 0,C 180,E1 11393.91,E2 11393.91} C_VEL
LIN {X 0,Y 183.405,Z 925.788,A -85,B 0,C 180,E1 11389.252,E2 11389.252} C_VEL
LIN {X 0,Y 196.07,Z 901.043,A -85,B 0,C 180,E1 11381.087,E2 11381.087} C_VEL
LIN {X 0,Y 209.235,Z 872.163,A -85,B 0,C 180,E1 11375.001,E2 11375.001} C_VEL
LIN {X 0,Y 220.706,Z 840.838,A -85,B 0,C 180,E1 11370.848,E2 11370.848} C_VEL
LIN {X 0,Y 224.78,Z 826.229,A -85,B 0,C 180,E1 11369.407,E2 11369.407} C_VEL
LIN {X 0,Y 218.87,Z 786.875,A -85,B 0,C 180,E1 11359.516,E2 11359.516} C_VEL
LIN {X 0,Y 214.075,Z 745.161,A -85,B 0,C 180,E1 11348.572,E2 11348.572} C_VEL
LIN {X 0,Y 212.067,Z 739.578,A -85,B 0,C 180,E1 11342.048,E2 11342.048} C_VEL
LIN {X 0,Y 212.138,Z 740.336,A -85,B 0,C 180,E1 11335.164,E2 11335.164} C_VEL
LIN {X 0,Y 215.515,Z 748.024,A -85,B 0,C 180,E1 11326.857,E2 11326.857} C_VEL
LIN {X 0,Y 220.29,Z 757.733,A -85,B 0,C 180,E1 11320.503,E2 11320.503} C_VEL
LIN {X 0,Y 226.513,Z 773.92,A -85,B 0,C 180,E1 11313.423,E2 11313.423} C_VEL
LIN {X 0,Y 230.86,Z 792.466,A -85,B 0,C 180,E1 11307.43,E2 11307.43} C_VEL
LIN {X 0,Y 231.993,Z 810.817,A -85,B 0,C 180,E1 11302.515,E2 11302.515} C_VEL
LIN {X 0,Y 220.179,Z 839.226,A -85,B 0,C 180,E1 11298.181,E2 11298.181} C_VEL
LIN {X 0,Y 206.813,Z 863.582,A -85,B 0,C 180,E1 11292.558,E2 11292.558} C_VEL
LIN {X 0,Y 192.886,Z 884.367,A -85,B 0,C 180,E1 11284.934,E2 11284.934} C_VEL
LIN {X 0,Y 181.506,Z 899.288,A -85,B 0,C 180,E1 11275.872,E2 11275.872} C_VEL
LIN {X 0,Y 173.666,Z 909.138,A -85,B 0,C 180,E1 11265.103,E2 11265.103} C_VEL
LIN {X 0,Y 170.522,Z 913.156,A -85,B 0,C 180,E1 11255.069,E2 11255.069} C_VEL
LIN {X 0,Y 170.516,Z 913.183,A -85,B 0,C 180,E1 11244.915,E2 11244.915} C_VEL
LIN {X 0,Y 173.66,Z 909.214,A -85,B 0,C 180,E1 11234.881,E2 11234.881} C_VEL
LIN {X 0,Y 181.49,Z 899.435,A -85,B 0,C 180,E1 11224.109,E2 11224.109} C_VEL
LIN {X 0,Y 192.693,Z 884.842,A -85,B 0,C 180,E1 11215.155,E2 11215.155} C_VEL
LIN {X 0,Y 206.614,Z 864.126,A -85,B 0,C 180,E1 11207.466,E2 11207.466} C_VEL
LIN {X 0,Y 220.12,Z 839.671,A -85,B 0,C 180,E1 11201.784,E2 11201.784} C_VEL
LIN {X 0,Y 223.347,Z 832.789,A -85,B 0,C 180,E1 11200.552,E2 11200.552} C_VEL
LIN {X 0,Y 223.288,Z 831.354,A -85,B 0,C 180,E1 11200.027,E2 11200.027} C_VEL
LIN {X 0,Y 200.26,Z 845.329,A -85,B 0,C 180,E1 11195.264,E2 11195.264} C_VEL
LIN {X 0,Y 181.319,Z 854.976,A -85,B 0,C 180,E1 11188.575,E2 11188.575} C_VEL
LIN {X 0,Y 179.021,Z 862.368,A -85,B 0,C 180,E1 11186.251,E2 11186.251} C_VEL
LIN {X 0,Y 173.502,Z 885.816,A -85,B 0,C 180,E1 11178.167,E2 11178.167} C_VEL
LIN {X 0,Y 170.531,Z 904.194,A -85,B 0,C 180,E1 11168.896,E2 11168.896} C_VEL
LIN {X 0,Y 170.965,Z 917.649,A -85,B 0,C 180,E1 11158.724,E2 11158.724} C_VEL
LIN {X 0,Y 175.966,Z 926.692,A -85,B 0,C 180,E1 11147.61,E2 11147.61} C_VEL
LIN {X 0,Y 188.22,Z 930.366,A -85,B 0,C 180,E1 11136.359,E2 11136.359} C_VEL
LIN {X 0,Y 203.098,Z 929.23,A -85,B 0,C 180,E1 11128.653,E2 11128.653} C_VEL
LIN {X 0,Y 213.37,Z 927.274,A -85,B 0,C 180,E1 11124.771,E2 11124.771} C_VEL
LIN {X 0,Y 208.686,Z 930.416,A -85,B 0,C 180,E1 11122.708,E2 11122.708} C_VEL
LIN {X 0,Y 179.77,Z 951.103,A -85,B 0,C 180,E1 11107.494,E2 11107.494} C_VEL
LIN {X 0,Y 169.587,Z 962.287,A -85,B 0,C 180,E1 11093.614,E2 11093.614} C_VEL
LIN {X 0,Y 167.774,Z 967.828,A -85,B 0,C 180,E1 11080.372,E2 11080.372} C_VEL
LIN {X 0,Y 169.117,Z 967.988,A -85,B 0,C 180,E1 11070.008,E2 11070.008} C_VEL
LIN {X 0,Y 168.287,Z 965.188,A -85,B 0,C 180,E1 11059.676,E2 11059.676} C_VEL
LIN {X 0,Y 169.302,Z 957.33,A -85,B 0,C 180,E1 11049.12,E2 11049.12} C_VEL
LIN {X 0,Y 174.732,Z 943.277,A -85,B 0,C 180,E1 11038.072,E2 11038.072} C_VEL
LIN {X 0,Y 183.405,Z 925.788,A -85,B 0,C 180,E1 11029.252,E2 11029.252} C_VEL
LIN {X 0,Y 185.324,Z 915.794,A -85,B 0,C 180,E1 11024.811,E2 11024.811} C_VEL
LIN {X 0,Y 187.92,Z 904.945,A -85,B 0,C 180,E1 11020.657,E2 11020.657} C_VEL
LIN {X 0,Y 201.72,Z 877.193,A -85,B 0,C 180,E1 11014.211,E2 11014.211} C_VEL
LIN {X 0,Y 213.811,Z 847.864,A -85,B 0,C 180,E1 11009.923,E2 11009.923} C_VEL
LIN {X 0,Y 219.614,Z 828.862,A -85,B 0,C 180,E1 11007.817,E2 11007.817} C_VEL
LIN {X 0,Y 215.477,Z 790.646,A -85,B 0,C 180,E1 10997.849,E2 10997.849} C_VEL
LIN {X 0,Y 212.591,Z 752.503,A -85,B 0,C 180,E1 10987.616,E2 10987.616} C_VEL
LIN {X 0,Y 210.952,Z 747.294,A -85,B 0,C 180,E1 10981.034,E2 10981.034} C_VEL
LIN {X 0,Y 211.111,Z 748.237,A -85,B 0,C 180,E1 10975.394,E2 10975.394} C_VEL
LIN {X 0,Y 214.007,Z 755.678,A -85,B 0,C 180,E1 10967.281,E2 10967.281} C_VEL
LIN {X 0,Y 218.081,Z 765.303,A -85,B 0,C 180,E1 10960.954,E2 10960.954} C_VEL
LIN {X 0,Y 222.819,Z 779.728,A -85,B 0,C 180,E1 10954.448,E2 10954.448} C_VEL
LIN {X 0,Y 226.19,Z 797.214,A -85,B 0,C 180,E1 10948.492,E2 10948.492} C_VEL
